LIN {X 0,Y 516.297,Z 411,A -85,B 0,C 180,E1 -4976.05,E2 -4976.05} C_VEL
LIN {X 0,Y 516.258,Z 415.654,A -85,B 0,C 180,E1 -4979.178,E2 -4979.178} C_VEL
LIN {X 0,Y 518.505,Z 428.002,A -85,B 0,C 180,E1 -4979.573,E2 -4979.573} C_VEL
LIN {X 0,Y 518.179,Z 441.043,A -85,B 0,C 180,E1 -4980.07,E2 -4980.07} C_VEL
LIN {X 0,Y 517.831,Z 453.233,A -85,B 0,C 180,E1 -4980.706,E2 -4980.706} C_VEL
LIN {X 0,Y 517.537,Z 464.053,A -85,B 0,C 180,E1 -4981.439,E2 -4981.439} C_VEL
LIN {X 0,Y 517.275,Z 474.235,A -85,B 0,C 180,E1 -4982.296,E2 -4982.296} C_VEL
LIN {X 0,Y 517.004,Z 483.822,A -85,B 0,C 180,E1 -4983.287,E2 -4983.287} C_VEL
LIN {X 0,Y 516.786,Z 492.252,A -85,B 0,C 180,E1 -4984.364,E2 -4984.364} C_VEL
LIN {X 0,Y 516.568,Z 499.577,A -85,B 0,C 180,E1 -4985.517,E2 -4985.517} C_VEL
LIN {X 0,Y 516.456,Z 505.994,A -85,B 0,C 180,E1 -4986.78,E2 -4986.78} C_VEL
LIN {X 0,Y 516.319,Z 511.794,A -85,B 0,C 180,E1 -4988.286,E2 -4988.286} C_VEL
LIN {X 0,Y 516.251,Z 515.814,A -85,B 0,C 180,E1 -4989.779,E2 -4989.779} C_VEL
LIN {X 0,Y 516.155,Z 517.667,A -85,B 0,C 180,E1 -4990.811,E2 -4990.811} C_VEL
LIN {X 0,Y 516.152,Z 518.842,A -85,B 0,C 180,E1 -4991.85,E2 -4991.85} C_VEL
LIN {X 0,Y 516.165,Z 519.286,A -85,B 0,C 180,E1 -4992.905,E2 -4992.905} C_VEL
LIN {X 0,Y 516.188,Z 519.003,A -85,B 0,C 180,E1 -4993.977,E2 -4993.977} C_VEL
LIN {X 0,Y 516.207,Z 517.97,A -85,B 0,C 180,E1 -4995.069,E2 -4995.069} C_VEL
LIN {X 0,Y 516.243,Z 516.116,A -85,B 0,C 180,E1 -4996.18,E2 -4996.18} C_VEL
LIN {X 0,Y 516.328,Z 512.006,A -85,B 0,C 180,E1 -4997.742,E2 -4997.742} C_VEL
LIN {X 0,Y 516.397,Z 508.021,A -85,B 0,C 180,E1 -4998.841,E2 -4998.841} C_VEL
LIN {X 0,Y 516.486,Z 502.965,A -85,B 0,C 180,E1 -4999.95,E2 -4999.95} C_VEL
LIN {X 0,Y 516.683,Z 495.416,A -85,B 0,C 180,E1 -5001.266,E2 -5001.266} C_VEL
LIN {X 0,Y 516.927,Z 487.189,A -85,B 0,C 180,E1 -5002.403,E2 -5002.403} C_VEL
LIN {X 0,Y 517.166,Z 478.617,A -85,B 0,C 180,E1 -5003.37,E2 -5003.37} C_VEL
LIN {X 0,Y 517.497,Z 467.836,A -85,B 0,C 180,E1 -5004.359,E2 -5004.359} C_VEL
LIN {X 0,Y 517.785,Z 457.319,A -85,B 0,C 180,E1 -5005.131,E2 -5005.131} C_VEL
LIN {X 0,Y 518.033,Z 446.537,A -85,B 0,C 180,E1 -5005.759,E2 -5005.759} C_VEL
LIN {X 0,Y 518.35,Z 433.197,A -85,B 0,C 180,E1 -5006.344,E2 -5006.344} C_VEL
LIN {X 0,Y 518.298,Z 426.521,A -85,B 0,C 180,E1 -5006.574,E2 -5006.574} C_VEL
LIN {X 0,Y 516.299,Z 415.747,A -85,B 0,C 180,E1 -5006.923,E2 -5006.923} C_VEL
LIN {X 0,Y 516.306,Z 411.528,A -85,B 0,C 180,E1 -5009.758,E2 -5009.758} C_VEL
LIN {X 0,Y 516.434,Z 407.634,A -85,B 0,C 180,E1 -5012.439,E2 -5012.439} C_VEL
LIN {X 0,Y 516.475,Z 403.919,A -85,B 0,C 180,E1 -5015.049,E2 -5015.049} C_VEL
LIN {X 0,Y 516.543,Z 400.144,A -85,B 0,C 180,E1 -5017.696,E2 -5017.696} C_VEL
LIN {X 0,Y 516.649,Z 396.744,A -85,B 0,C 180,E1 -5020.118,E2 -5020.118} C_VEL
LIN {X 0,Y 516.675,Z 393.324,A -85,B 0,C 180,E1 -5022.587,E2 -5022.587} C_VEL
LIN {X 0,Y 516.733,Z 388.827,A -85,B 0,C 180,E1 -5025.829,E2 -5025.829} C_VEL
LIN {X 0,Y 516.781,Z 386.668,A -85,B 0,C 180,E1 -5027.432,E2 -5027.432} C_VEL
LIN {X 0,Y 516.874,Z 386.105,A -85,B 0,C 180,E1 -5028.232,E2 -5028.232} C_VEL
LIN {X 0,Y 516.968,Z 386.095,A -85,B 0,C 180,E1 -5031.4,E2 -5031.4} C_VEL
LIN {X 0,Y 517.006,Z 386.087,A -85,B 0,C 180,E1 -5033.757,E2 -5033.757} C_VEL
LIN {X 0,Y 517.079,Z 386.08,A -85,B 0,C 180,E1 -5037.663,E2 -5037.663} C_VEL
LIN {X 0,Y 517.092,Z 386.078,A -85,B 0,C 180,E1 -5040.779,E2 -5040.779} C_VEL
LIN {X 0,Y 517.01,Z 386.086,A -85,B 0,C 180,E1 -5043.117,E2 -5043.117} C_VEL
LIN {X 0,Y 517.008,Z 386.087,A -85,B 0,C 180,E1 -5046.243,E2 -5046.243} C_VEL
LIN {X 0,Y 516.951,Z 386.093,A -85,B 0,C 180,E1 -5049.389,E2 -5049.389} C_VEL
LIN {X 0,Y 516.948,Z 386.094,A -85,B 0,C 180,E1 -5051.808,E2 -5051.808} C_VEL
LIN {X 0,Y 516.94,Z 386.096,A -85,B 0,C 180,E1 -5055.147,E2 -5055.147} C_VEL
LIN {X 0,Y 516.922,Z 386.098,A -85,B 0,C 180,E1 -5058.222,E2 -5058.222} C_VEL
LIN {X 0,Y 516.91,Z 386.099,A -85,B 0,C 180,E1 -5060.702,E2 -5060.702} C_VEL
LIN {X 0,Y 516.908,Z 386.097,A -85,B 0,C 180,E1 -5064.072,E2 -5064.072} C_VEL
LIN {X 0,Y 516.926,Z 386.098,A -85,B 0,C 180,E1 -5066.658,E2 -5066.658} C_VEL
LIN {X 0,Y 516.922,Z 386.097,A -85,B 0,C 180,E1 -5069.527,E2 -5069.527} C_VEL
LIN {X 0,Y 516.895,Z 386.1,A -85,B 0,C 180,E1 -5072.544,E2 -5072.544} C_VEL
LIN {X 0,Y 516.878,Z 386.103,A -85,B 0,C 180,E1 -5075.333,E2 -5075.333} C_VEL
LIN {X 0,Y 516.88,Z 386.104,A -85,B 0,C 180,E1 -5077.944,E2 -5077.944} C_VEL
LIN {X 0,Y 516.902,Z 386.1,A -85,B 0,C 180,E1 -5080.74,E2 -5080.74} C_VEL
LIN {X 0,Y 516.881,Z 386.103,A -85,B 0,C 180,E1 -5083.904,E2 -5083.904} C_VEL
LIN {X 0,Y 516.88,Z 386.102,A -85,B 0,C 180,E1 -5086.108,E2 -5086.108} C_VEL
LIN {X 0,Y 516.903,Z 386.1,A -85,B 0,C 180,E1 -5089.261,E2 -5089.261} C_VEL
LIN {X 0,Y 516.918,Z 386.26,A -85,B 0,C 180,E1 -5091.913,E2 -5091.913} C_VEL
LIN {X 0,Y 517.626,Z 390.379,A -85,B 0,C 180,E1 -5093.8,E2 -5093.8} C_VEL
LIN {X 0,Y 517.687,Z 395.366,A -85,B 0,C 180,E1 -5095.907,E2 -5095.907} C_VEL
LIN {X 0,Y 517.366,Z 402.877,A -85,B 0,C 180,E1 -5098.923,E2 -5098.923} C_VEL
LIN {X 0,Y 517.163,Z 409.885,A -85,B 0,C 180,E1 -5101.6,E2 -5101.6} C_VEL
LIN {X 0,Y 516.952,Z 418.116,A -85,B 0,C 180,E1 -5104.644,E2 -5104.644} C_VEL
LIN {X 0,Y 516.833,Z 426.501,A -85,B 0,C 180,E1 -5107.62,E2 -5107.62} C_VEL
LIN {X 0,Y 516.682,Z 434.848,A -85,B 0,C 180,E1 -5110.534,E2 -5110.534} C_VEL
LIN {X 0,Y 516.553,Z 443.402,A -85,B 0,C 180,E1 -5113.399,E2 -5113.399} C_VEL
LIN {X 0,Y 516.494,Z 451.498,A -85,B 0,C 180,E1 -5116.099,E2 -5116.099} C_VEL
LIN {X 0,Y 518.453,Z 465.116,A -85,B 0,C 180,E1 -5116.477,E2 -5116.477} C_VEL
LIN {X 0,Y 518.192,Z 477.346,A -85,B 0,C 180,E1 -5116.92,E2 -5116.92} C_VEL
LIN {X 0,Y 517.871,Z 489.784,A -85,B 0,C 180,E1 -5117.534,E2 -5117.534} C_VEL
LIN {X 0,Y 517.617,Z 500.953,A -85,B 0,C 180,E1 -5118.249,E2 -5118.249} C_VEL
LIN {X 0,Y 517.316,Z 511.907,A -85,B 0,C 180,E1 -5119.135,E2 -5119.135} C_VEL
LIN {X 0,Y 517.003,Z 520.836,A -85,B 0,C 180,E1 -5120.019,E2 -5120.019} C_VEL
LIN {X 0,Y 516.755,Z 530.543,A -85,B 0,C 180,E1 -5121.199,E2 -5121.199} C_VEL
LIN {X 0,Y 516.562,Z 538.27,A -85,B 0,C 180,E1 -5122.377,E2 -5122.377} C_VEL
LIN {X 0,Y 516.427,Z 545.391,A -85,B 0,C 180,E1 -5123.75,E2 -5123.75} C_VEL
LIN {X 0,Y 516.313,Z 550.128,A -85,B 0,C 180,E1 -5124.924,E2 -5124.924} C_VEL
LIN {X 0,Y 516.355,Z 553.751,A -85,B 0,C 180,E1 -5126.098,E2 -5126.098} C_VEL
LIN {X 0,Y 516.282,Z 555.616,A -85,B 0,C 180,E1 -5126.879,E2 -5126.879} C_VEL
LIN {X 0,Y 516.261,Z 557.015,A -85,B 0,C 180,E1 -5127.66,E2 -5127.66} C_VEL
LIN {X 0,Y 516.16,Z 558.621,A -85,B 0,C 180,E1 -5129.22,E2 -5129.22} C_VEL
LIN {X 0,Y 516.154,Z 558.838,A -85,B 0,C 180,E1 -5130,E2 -5130} C_VEL
LIN {X 0,Y 516.192,Z 558.015,A -85,B 0,C 180,E1 -5131.561,E2 -5131.561} C_VEL
LIN {X 0,Y 516.261,Z 557.021,A -85,B 0,C 180,E1 -5132.341,E2 -5132.341} C_VEL
LIN {X 0,Y 516.282,Z 555.624,A -85,B 0,C 180,E1 -5133.122,E2 -5133.122} C_VEL
LIN {X 0,Y 516.326,Z 552.683,A -85,B 0,C 180,E1 -5134.294,E2 -5134.294} C_VEL
LIN {X 0,Y 516.383,Z 548.702,A -85,B 0,C 180,E1 -5135.467,E2 -5135.467} C_VEL
LIN {X 0,Y 516.465,Z 543.401,A -85,B 0,C 180,E1 -5136.679,E2 -5136.679} C_VEL
LIN {X 0,Y 516.598,Z 537.125,A -85,B 0,C 180,E1 -5137.819,E2 -5137.819} C_VEL
LIN {X 0,Y 516.807,Z 529.078,A -85,B 0,C 180,E1 -5138.997,E2 -5138.997} C_VEL
LIN {X 0,Y 516.999,Z 520.876,A -85,B 0,C 180,E1 -5139.981,E2 -5139.981} C_VEL
LIN {X 0,Y 517.318,Z 510.879,A -85,B 0,C 180,E1 -5140.964,E2 -5140.964} C_VEL
LIN {X 0,Y 517.612,Z 501.016,A -85,B 0,C 180,E1 -5141.752,E2 -5141.752} C_VEL
LIN {X 0,Y 517.849,Z 489.862,A -85,B 0,C 180,E1 -5142.467,E2 -5142.467} C_VEL
LIN {X 0,Y 518.17,Z 477.41,A -85,B 0,C 180,E1 -5143.082,E2 -5143.082} C_VEL
LIN {X 0,Y 518.465,Z 464.339,A -85,B 0,C 180,E1 -5143.548,E2 -5143.548} C_VEL
LIN {X 0,Y 516.493,Z 451.65,A -85,B 0,C 180,E1 -5143.902,E2 -5143.902} C_VEL
LIN {X 0,Y 516.597,Z 442.444,A -85,B 0,C 180,E1 -5147.008,E2 -5147.008} C_VEL
LIN {X 0,Y 516.704,Z 433.963,A -85,B 0,C 180,E1 -5149.879,E2 -5149.879} C_VEL
LIN {X 0,Y 516.859,Z 425.579,A -85,B 0,C 180,E1 -5152.801,E2 -5152.801} C_VEL
LIN {X 0,Y 517.023,Z 417.316,A -85,B 0,C 180,E1 -5155.784,E2 -5155.784} C_VEL
LIN {X 0,Y 517.18,Z 410.238,A -85,B 0,C 180,E1 -5158.4,E2 -5158.4} C_VEL
LIN {X 0,Y 517.389,Z 403.001,A -85,B 0,C 180,E1 -5161.155,E2 -5161.155} C_VEL
LIN {X 0,Y 517.701,Z 395.519,A -85,B 0,C 180,E1 -5164.096,E2 -5164.096} C_VEL
LIN {X 0,Y 517.747,Z 391.578,A -85,B 0,C 180,E1 -5165.711,E2 -5165.711} C_VEL
LIN {X 0,Y 516.892,Z 386.102,A -85,B 0,C 180,E1 -5168.088,E2 -5168.088} C_VEL
LIN {X 0,Y 516.886,Z 386.102,A -85,B 0,C 180,E1 -5170.741,E2 -5170.741} C_VEL
LIN {X 0,Y 516.884,Z 386.101,A -85,B 0,C 180,E1 -5172.831,E2 -5172.831} C_VEL
LIN {X 0,Y 516.896,Z 386.101,A -85,B 0,C 180,E1 -5175.007,E2 -5175.007} C_VEL
LIN {X 0,Y 516.914,Z 386.098,A -85,B 0,C 180,E1 -5178.399,E2 -5178.399} C_VEL
LIN {X 0,Y 516.882,Z 386.101,A -85,B 0,C 180,E1 -5181.284,E2 -5181.284} C_VEL
LIN {X 0,Y 516.887,Z 386.101,A -85,B 0,C 180,E1 -5184.221,E2 -5184.221} C_VEL
LIN {X 0,Y 516.895,Z 386.1,A -85,B 0,C 180,E1 -5187.457,E2 -5187.457} C_VEL
LIN {X 0,Y 516.922,Z 386.096,A -85,B 0,C 180,E1 -5190.695,E2 -5190.695} C_VEL
LIN {X 0,Y 516.943,Z 386.095,A -85,B 0,C 180,E1 -5193.804,E2 -5193.804} C_VEL
LIN {X 0,Y 516.866,Z 386.103,A -85,B 0,C 180,E1 -5196.776,E2 -5196.776} C_VEL
LIN {X 0,Y 516.94,Z 386.095,A -85,B 0,C 180,E1 -5199.732,E2 -5199.732} C_VEL
LIN {X 0,Y 516.922,Z 386.096,A -85,B 0,C 180,E1 -5202.596,E2 -5202.596} C_VEL
LIN {X 0,Y 516.943,Z 386.094,A -85,B 0,C 180,E1 -5205.03,E2 -5205.03} C_VEL
LIN {X 0,Y 516.966,Z 386.092,A -85,B 0,C 180,E1 -5208.234,E2 -5208.234} C_VEL
LIN {X 0,Y 516.97,Z 386.091,A -85,B 0,C 180,E1 -5211.4,E2 -5211.4} C_VEL
LIN {X 0,Y 517.011,Z 386.086,A -85,B 0,C 180,E1 -5213.757,E2 -5213.757} C_VEL
LIN {X 0,Y 517.082,Z 386.077,A -85,B 0,C 180,E1 -5217.663,E2 -5217.663} C_VEL
LIN {X 0,Y 517.093,Z 386.075,A -85,B 0,C 180,E1 -5220.779,E2 -5220.779} C_VEL
LIN {X 0,Y 517.014,Z 386.085,A -85,B 0,C 180,E1 -5223.117,E2 -5223.117} C_VEL
LIN {X 0,Y 517.011,Z 386.087,A -85,B 0,C 180,E1 -5226.243,E2 -5226.243} C_VEL
LIN {X 0,Y 516.953,Z 386.094,A -85,B 0,C 180,E1 -5229.389,E2 -5229.389} C_VEL
LIN {X 0,Y 516.952,Z 386.093,A -85,B 0,C 180,E1 -5231.807,E2 -5231.807} C_VEL
LIN {X 0,Y 516.945,Z 386.094,A -85,B 0,C 180,E1 -5235.146,E2 -5235.146} C_VEL
LIN {X 0,Y 516.926,Z 386.097,A -85,B 0,C 180,E1 -5238.222,E2 -5238.222} C_VEL
LIN {X 0,Y 516.912,Z 386.098,A -85,B 0,C 180,E1 -5240.701,E2 -5240.701} C_VEL
LIN {X 0,Y 516.904,Z 386.1,A -85,B 0,C 180,E1 -5244.072,E2 -5244.072} C_VEL
LIN {X 0,Y 516.926,Z 386.096,A -85,B 0,C 180,E1 -5246.658,E2 -5246.658} C_VEL
LIN {X 0,Y 516.911,Z 386.098,A -85,B 0,C 180,E1 -5249.524,E2 -5249.524} C_VEL
LIN {X 0,Y 516.898,Z 386.1,A -85,B 0,C 180,E1 -5252.544,E2 -5252.544} C_VEL
LIN {X 0,Y 516.881,Z 386.101,A -85,B 0,C 180,E1 -5255.332,E2 -5255.332} C_VEL
LIN {X 0,Y 516.882,Z 386.101,A -85,B 0,C 180,E1 -5257.943,E2 -5257.943} C_VEL
LIN {X 0,Y 516.883,Z 386.103,A -85,B 0,C 180,E1 -5260.742,E2 -5260.742} C_VEL
LIN {X 0,Y 516.885,Z 386.103,A -85,B 0,C 180,E1 -5262.831,E2 -5262.831} C_VEL
LIN {X 0,Y 516.896,Z 386.1,A -85,B 0,C 180,E1 -5265.007,E2 -5265.007} C_VEL
LIN {X 0,Y 516.918,Z 386.097,A -85,B 0,C 180,E1 -5268.398,E2 -5268.398} C_VEL
LIN {X 0,Y 516.882,Z 386.103,A -85,B 0,C 180,E1 -5270.296,E2 -5270.296} C_VEL
LIN {X 0,Y 516.211,Z 386.186,A -85,B 0,C 180,E1 -5270.946,E2 -5270.946} C_VEL
LIN {X 0,Y 513.366,Z 386.54,A -85,B 0,C 180,E1 -5272.002,E2 -5272.002} C_VEL
LIN {X 0,Y 510.96,Z 386.841,A -85,B 0,C 180,E1 -5272.852,E2 -5272.852} C_VEL
LIN {X 0,Y 509.92,Z 386.97,A -85,B 0,C 180,E1 -5273.509,E2 -5273.509} C_VEL
LIN {X 0,Y 509.832,Z 386.979,A -85,B 0,C 180,E1 -5273.731,E2 -5273.731} C_VEL
LIN {X 0,Y 509.862,Z 386.976,A -85,B 0,C 180,E1 -5276.539,E2 -5276.539} C_VEL
LIN {X 0,Y 509.847,Z 386.978,A -85,B 0,C 180,E1 -5279.334,E2 -5279.334} C_VEL
LIN {X 0,Y 509.894,Z 386.973,A -85,B 0,C 180,E1 -5282.054,E2 -5282.054} C_VEL
LIN {X 0,Y 509.879,Z 386.974,A -85,B 0,C 180,E1 -5284.704,E2 -5284.704} C_VEL
LIN {X 0,Y 509.829,Z 386.978,A -85,B 0,C 180,E1 -5287.458,E2 -5287.458} C_VEL
LIN {X 0,Y 509.919,Z 386.968,A -85,B 0,C 180,E1 -5289.845,E2 -5289.845} C_VEL
LIN {X 0,Y 509.881,Z 386.972,A -85,B 0,C 180,E1 -5293.174,E2 -5293.174} C_VEL
LIN {X 0,Y 509.866,Z 386.975,A -85,B 0,C 180,E1 -5295.634,E2 -5295.634} C_VEL
LIN {X 0,Y 509.915,Z 386.969,A -85,B 0,C 180,E1 -5298.874,E2 -5298.874} C_VEL
LIN {X 0,Y 509.953,Z 386.965,A -85,B 0,C 180,E1 -5302.078,E2 -5302.078} C_VEL
LIN {X 0,Y 509.984,Z 386.962,A -85,B 0,C 180,E1 -5304.464,E2 -5304.464} C_VEL
LIN {X 0,Y 510.058,Z 386.951,A -85,B 0,C 180,E1 -5307.631,E2 -5307.631} C_VEL
LIN {X 0,Y 510.066,Z 386.951,A -85,B 0,C 180,E1 -5310.789,E2 -5310.789} C_VEL
LIN {X 0,Y 509.956,Z 386.964,A -85,B 0,C 180,E1 -5313.16,E2 -5313.16} C_VEL
LIN {X 0,Y 509.938,Z 386.967,A -85,B 0,C 180,E1 -5316.33,E2 -5316.33} C_VEL
LIN {X 0,Y 509.706,Z 386.998,A -85,B 0,C 180,E1 -5318.723,E2 -5318.723} C_VEL
LIN {X 0,Y 509.616,Z 391.348,A -85,B 0,C 180,E1 -5321.938,E2 -5321.938} C_VEL
LIN {X 0,Y 509.499,Z 395.893,A -85,B 0,C 180,E1 -5325.193,E2 -5325.193} C_VEL
LIN {X 0,Y 509.404,Z 400.582,A -85,B 0,C 180,E1 -5328.5,E2 -5328.5} C_VEL
LIN {X 0,Y 509.281,Z 404.229,A -85,B 0,C 180,E1 -5331.026,E2 -5331.026} C_VEL
LIN {X 0,Y 509.258,Z 407.951,A -85,B 0,C 180,E1 -5333.591,E2 -5333.591} C_VEL
LIN {X 0,Y 509.213,Z 411.861,A -85,B 0,C 180,E1 -5336.219,E2 -5336.219} C_VEL
LIN {X 0,Y 509.193,Z 416.037,A -85,B 0,C 180,E1 -5338.997,E2 -5338.997} C_VEL
LIN {X 0,Y 511.576,Z 428.689,A -85,B 0,C 180,E1 -5339.404,E2 -5339.404} C_VEL
LIN {X 0,Y 511.235,Z 441.825,A -85,B 0,C 180,E1 -5339.916,E2 -5339.916} C_VEL
LIN {X 0,Y 510.919,Z 453.048,A -85,B 0,C 180,E1 -5340.511,E2 -5340.511} C_VEL
LIN {X 0,Y 510.566,Z 464.641,A -85,B 0,C 180,E1 -5341.307,E2 -5341.307} C_VEL
LIN {X 0,Y 510.273,Z 475.615,A -85,B 0,C 180,E1 -5342.255,E2 -5342.255} C_VEL
LIN {X 0,Y 509.992,Z 485.086,A -85,B 0,C 180,E1 -5343.275,E2 -5343.275} C_VEL
LIN {X 0,Y 509.718,Z 493.709,A -85,B 0,C 180,E1 -5344.423,E2 -5344.423} C_VEL
LIN {X 0,Y 509.497,Z 501.397,A -85,B 0,C 180,E1 -5345.694,E2 -5345.694} C_VEL
LIN {X 0,Y 509.314,Z 507.926,A -85,B 0,C 180,E1 -5347.087,E2 -5347.087} C_VEL
LIN {X 0,Y 509.235,Z 512.588,A -85,B 0,C 180,E1 -5348.392,E2 -5348.392} C_VEL
LIN {X 0,Y 509.14,Z 516.501,A -85,B 0,C 180,E1 -5349.931,E2 -5349.931} C_VEL
LIN {X 0,Y 509.058,Z 518.806,A -85,B 0,C 180,E1 -5351.504,E2 -5351.504} C_VEL
LIN {X 0,Y 509.079,Z 519.572,A -85,B 0,C 180,E1 -5352.972,E2 -5352.972} C_VEL
LIN {X 0,Y 509.105,Z 519.195,A -85,B 0,C 180,E1 -5354.123,E2 -5354.123} C_VEL
LIN {X 0,Y 509.121,Z 518.028,A -85,B 0,C 180,E1 -5355.25,E2 -5355.25} C_VEL
LIN {X 0,Y 509.173,Z 516.09,A -85,B 0,C 180,E1 -5356.359,E2 -5356.359} C_VEL
LIN {X 0,Y 509.271,Z 512.167,A -85,B 0,C 180,E1 -5357.843,E2 -5357.843} C_VEL
LIN {X 0,Y 509.324,Z 508.083,A -85,B 0,C 180,E1 -5358.974,E2 -5358.974} C_VEL
LIN {X 0,Y 509.487,Z 501.648,A -85,B 0,C 180,E1 -5360.359,E2 -5360.359} C_VEL
LIN {X 0,Y 509.705,Z 493.893,A -85,B 0,C 180,E1 -5361.649,E2 -5361.649} C_VEL
LIN {X 0,Y 509.967,Z 486.313,A -85,B 0,C 180,E1 -5362.672,E2 -5362.672} C_VEL
LIN {X 0,Y 510.244,Z 477.233,A -85,B 0,C 180,E1 -5363.681,E2 -5363.681} C_VEL
LIN {X 0,Y 510.569,Z 467.144,A -85,B 0,C 180,E1 -5364.594,E2 -5364.594} C_VEL
LIN {X 0,Y 510.863,Z 456.701,A -85,B 0,C 180,E1 -5365.352,E2 -5365.352} C_VEL
LIN {X 0,Y 511.157,Z 444.61,A -85,B 0,C 180,E1 -5366.044,E2 -5366.044} C_VEL
LIN {X 0,Y 511.464,Z 433.096,A -85,B 0,C 180,E1 -5366.54,E2 -5366.54} C_VEL
LIN {X 0,Y 511.261,Z 426.599,A -85,B 0,C 180,E1 -5366.768,E2 -5366.768} C_VEL
LIN {X 0,Y 509.233,Z 416.078,A -85,B 0,C 180,E1 -5367.1,E2 -5367.1} C_VEL
LIN {X 0,Y 509.269,Z 411.267,A -85,B 0,C 180,E1 -5370.389,E2 -5370.389} C_VEL
LIN {X 0,Y 509.34,Z 407.659,A -85,B 0,C 180,E1 -5372.913,E2 -5372.913} C_VEL
LIN {X 0,Y 509.413,Z 403.837,A -85,B 0,C 180,E1 -5375.58,E2 -5375.58} C_VEL
LIN {X 0,Y 509.486,Z 400.261,A -85,B 0,C 180,E1 -5378.133,E2 -5378.133} C_VEL
LIN {X 0,Y 509.561,Z 396.743,A -85,B 0,C 180,E1 -5380.67,E2 -5380.67} C_VEL
LIN {X 0,Y 509.604,Z 393.284,A -85,B 0,C 180,E1 -5383.165,E2 -5383.165} C_VEL
LIN {X 0,Y 509.698,Z 389.968,A -85,B 0,C 180,E1 -5385.629,E2 -5385.629} C_VEL
LIN {X 0,Y 509.722,Z 387.777,A -85,B 0,C 180,E1 -5387.255,E2 -5387.255} C_VEL
LIN {X 0,Y 509.822,Z 386.984,A -85,B 0,C 180,E1 -5388.164,E2 -5388.164} C_VEL
LIN {X 0,Y 509.914,Z 386.974,A -85,B 0,C 180,E1 -5391.28,E2 -5391.28} C_VEL
LIN {X 0,Y 509.974,Z 386.963,A -85,B 0,C 180,E1 -5393.67,E2 -5393.67} C_VEL
LIN {X 0,Y 510.051,Z 386.955,A -85,B 0,C 180,E1 -5397.631,E2 -5397.631} C_VEL
LIN {X 0,Y 510.062,Z 386.953,A -85,B 0,C 180,E1 -5400.79,E2 -5400.79} C_VEL
LIN {X 0,Y 509.952,Z 386.965,A -85,B 0,C 180,E1 -5403.16,E2 -5403.16} C_VEL
LIN {X 0,Y 509.976,Z 386.962,A -85,B 0,C 180,E1 -5406.33,E2 -5406.33} C_VEL
LIN {X 0,Y 509.912,Z 386.97,A -85,B 0,C 180,E1 -5408.72,E2 -5408.72} C_VEL
LIN {X 0,Y 509.9,Z 386.972,A -85,B 0,C 180,E1 -5411.932,E2 -5411.932} C_VEL
LIN {X 0,Y 509.889,Z 386.975,A -85,B 0,C 180,E1 -5415.242,E2 -5415.242} C_VEL
LIN {X 0,Y 509.885,Z 386.973,A -85,B 0,C 180,E1 -5418.001,E2 -5418.001} C_VEL
LIN {X 0,Y 509.848,Z 386.978,A -85,B 0,C 180,E1 -5421.002,E2 -5421.002} C_VEL
LIN {X 0,Y 509.833,Z 386.981,A -85,B 0,C 180,E1 -5423.563,E2 -5423.563} C_VEL
LIN {X 0,Y 509.91,Z 386.97,A -85,B 0,C 180,E1 -5426.38,E2 -5426.38} C_VEL
LIN {X 0,Y 509.883,Z 386.976,A -85,B 0,C 180,E1 -5428.844,E2 -5428.844} C_VEL
LIN {X 0,Y 509.819,Z 386.982,A -85,B 0,C 180,E1 -5431.59,E2 -5431.59} C_VEL
LIN {X 0,Y 509.85,Z 386.978,A -85,B 0,C 180,E1 -5434.414,E2 -5434.414} C_VEL
LIN {X 0,Y 509.817,Z 386.984,A -85,B 0,C 180,E1 -5437.341,E2 -5437.341} C_VEL
LIN {X 0,Y 509.86,Z 386.979,A -85,B 0,C 180,E1 -5440.38,E2 -5440.38} C_VEL
LIN {X 0,Y 509.822,Z 386.982,A -85,B 0,C 180,E1 -5443.063,E2 -5443.063} C_VEL
LIN {X 0,Y 509.828,Z 386.981,A -85,B 0,C 180,E1 -5445.793,E2 -5445.793} C_VEL
LIN {X 0,Y 509.865,Z 386.975,A -85,B 0,C 180,E1 -5448.576,E2 -5448.576} C_VEL
LIN {X 0,Y 509.854,Z 387.091,A -85,B 0,C 180,E1 -5451.663,E2 -5451.663} C_VEL
LIN {X 0,Y 510.636,Z 391.477,A -85,B 0,C 180,E1 -5453.715,E2 -5453.715} C_VEL
LIN {X 0,Y 510.706,Z 395.971,A -85,B 0,C 180,E1 -5455.658,E2 -5455.658} C_VEL
LIN {X 0,Y 510.391,Z 403.245,A -85,B 0,C 180,E1 -5458.62,E2 -5458.62} C_VEL
LIN {X 0,Y 510.167,Z 409.74,A -85,B 0,C 180,E1 -5461.174,E2 -5461.174} C_VEL
LIN {X 0,Y 509.949,Z 417.958,A -85,B 0,C 180,E1 -5464.271,E2 -5464.271} C_VEL
LIN {X 0,Y 509.778,Z 426.769,A -85,B 0,C 180,E1 -5467.472,E2 -5467.472} C_VEL
LIN {X 0,Y 509.609,Z 434.653,A -85,B 0,C 180,E1 -5470.253,E2 -5470.253} C_VEL
LIN {X 0,Y 509.485,Z 443.148,A -85,B 0,C 180,E1 -5473.162,E2 -5473.162} C_VEL
LIN {X 0,Y 509.395,Z 451.195,A -85,B 0,C 180,E1 -5475.901,E2 -5475.901} C_VEL
LIN {X 0,Y 511.524,Z 465.534,A -85,B 0,C 180,E1 -5476.316,E2 -5476.316} C_VEL
LIN {X 0,Y 511.24,Z 478.133,A -85,B 0,C 180,E1 -5476.789,E2 -5476.789} C_VEL
LIN {X 0,Y 510.887,Z 490.799,A -85,B 0,C 180,E1 -5477.438,E2 -5477.438} C_VEL
LIN {X 0,Y 510.605,Z 501.947,A -85,B 0,C 180,E1 -5478.186,E2 -5478.186} C_VEL
LIN {X 0,Y 510.285,Z 512.66,A -85,B 0,C 180,E1 -5479.084,E2 -5479.084} C_VEL
LIN {X 0,Y 509.937,Z 522.316,A -85,B 0,C 180,E1 -5480.08,E2 -5480.08} C_VEL
LIN {X 0,Y 509.703,Z 530.235,A -85,B 0,C 180,E1 -5481.077,E2 -5481.077} C_VEL
LIN {X 0,Y 509.494,Z 537.971,A -85,B 0,C 180,E1 -5482.271,E2 -5482.271} C_VEL
LIN {X 0,Y 509.326,Z 545.098,A -85,B 0,C 180,E1 -5483.663,E2 -5483.663} C_VEL
LIN {X 0,Y 509.245,Z 549.842,A -85,B 0,C 180,E1 -5484.854,E2 -5484.854} C_VEL
LIN {X 0,Y 509.25,Z 553.468,A -85,B 0,C 180,E1 -5486.044,E2 -5486.044} C_VEL
LIN {X 0,Y 509.2,Z 555.338,A -85,B 0,C 180,E1 -5486.836,E2 -5486.836} C_VEL
LIN {X 0,Y 509.19,Z 556.74,A -85,B 0,C 180,E1 -5487.627,E2 -5487.627} C_VEL
LIN {X 0,Y 509.073,Z 558.348,A -85,B 0,C 180,E1 -5489.209,E2 -5489.209} C_VEL
LIN {X 0,Y 509.065,Z 558.567,A -85,B 0,C 180,E1 -5490,E2 -5490} C_VEL
LIN {X 0,Y 509.112,Z 557.745,A -85,B 0,C 180,E1 -5491.582,E2 -5491.582} C_VEL
LIN {X 0,Y 509.19,Z 556.752,A -85,B 0,C 180,E1 -5492.373,E2 -5492.373} C_VEL
LIN {X 0,Y 509.201,Z 555.353,A -85,B 0,C 180,E1 -5493.165,E2 -5493.165} C_VEL
LIN {X 0,Y 509.216,Z 552.411,A -85,B 0,C 180,E1 -5494.354,E2 -5494.354} C_VEL
LIN {X 0,Y 509.305,Z 548.43,A -85,B 0,C 180,E1 -5495.543,E2 -5495.543} C_VEL
LIN {X 0,Y 509.402,Z 542.757,A -85,B 0,C 180,E1 -5496.845,E2 -5496.845} C_VEL
LIN {X 0,Y 509.563,Z 535.606,A -85,B 0,C 180,E1 -5498.127,E2 -5498.127} C_VEL
LIN {X 0,Y 509.793,Z 527.301,A -85,B 0,C 180,E1 -5499.322,E2 -5499.322} C_VEL
LIN {X 0,Y 510.013,Z 518.782,A -85,B 0,C 180,E1 -5500.32,E2 -5500.32} C_VEL
LIN {X 0,Y 510.406,Z 508.264,A -85,B 0,C 180,E1 -5501.316,E2 -5501.316} C_VEL
LIN {X 0,Y 510.66,Z 497.108,A -85,B 0,C 180,E1 -5502.168,E2 -5502.168} C_VEL
LIN {X 0,Y 511.004,Z 486.461,A -85,B 0,C 180,E1 -5502.813,E2 -5502.813} C_VEL
LIN {X 0,Y 511.327,Z 474.749,A -85,B 0,C 180,E1 -5503.361,E2 -5503.361} C_VEL
LIN {X 0,Y 511.34,Z 463.555,A -85,B 0,C 180,E1 -5503.753,E2 -5503.753} C_VEL
LIN {X 0,Y 509.404,Z 451.39,A -85,B 0,C 180,E1 -5504.099,E2 -5504.099} C_VEL
LIN {X 0,Y 509.499,Z 443.469,A -85,B 0,C 180,E1 -5506.839,E2 -5506.839} C_VEL
LIN {X 0,Y 509.647,Z 434.994,A -85,B 0,C 180,E1 -5509.746,E2 -5509.746} C_VEL
LIN {X 0,Y 509.81,Z 426.62,A -85,B 0,C 180,E1 -5512.706,E2 -5512.706} C_VEL
LIN {X 0,Y 509.985,Z 418.367,A -85,B 0,C 180,E1 -5515.728,E2 -5515.728} C_VEL
LIN {X 0,Y 510.185,Z 410.121,A -85,B 0,C 180,E1 -5518.825,E2 -5518.825} C_VEL
LIN {X 0,Y 510.419,Z 403.092,A -85,B 0,C 180,E1 -5521.549,E2 -5521.549} C_VEL
LIN {X 0,Y 510.73,Z 396.125,A -85,B 0,C 180,E1 -5524.346,E2 -5524.346} C_VEL
LIN {X 0,Y 510.595,Z 391.497,A -85,B 0,C 180,E1 -5526.29,E2 -5526.29} C_VEL
LIN {X 0,Y 509.855,Z 386.978,A -85,B 0,C 180,E1 -5528.338,E2 -5528.338} C_VEL
LIN {X 0,Y 509.859,Z 386.977,A -85,B 0,C 180,E1 -5531.425,E2 -5531.425} C_VEL
LIN {X 0,Y 509.84,Z 386.98,A -85,B 0,C 180,E1 -5534.67,E2 -5534.67} C_VEL
LIN {X 0,Y 509.857,Z 386.977,A -85,B 0,C 180,E1 -5538.103,E2 -5538.103} C_VEL
LIN {X 0,Y 509.847,Z 386.978,A -85,B 0,C 180,E1 -5540.647,E2 -5540.647} C_VEL
LIN {X 0,Y 509.835,Z 386.979,A -85,B 0,C 180,E1 -5543.647,E2 -5543.647} C_VEL
LIN {X 0,Y 509.843,Z 386.978,A -85,B 0,C 180,E1 -5546.538,E2 -5546.538} C_VEL
LIN {X 0,Y 509.846,Z 386.978,A -85,B 0,C 180,E1 -5549.334,E2 -5549.334} C_VEL
LIN {X 0,Y 509.893,Z 386.97,A -85,B 0,C 180,E1 -5552.054,E2 -5552.054} C_VEL
LIN {X 0,Y 509.877,Z 386.974,A -85,B 0,C 180,E1 -5554.704,E2 -5554.704} C_VEL
LIN {X 0,Y 509.827,Z 386.981,A -85,B 0,C 180,E1 -5557.458,E2 -5557.458} C_VEL
LIN {X 0,Y 509.917,Z 386.969,A -85,B 0,C 180,E1 -5559.845,E2 -5559.845} C_VEL
LIN {X 0,Y 509.882,Z 386.975,A -85,B 0,C 180,E1 -5563.175,E2 -5563.175} C_VEL
LIN {X 0,Y 509.864,Z 386.977,A -85,B 0,C 180,E1 -5565.634,E2 -5565.634} C_VEL
LIN {X 0,Y 509.913,Z 386.97,A -85,B 0,C 180,E1 -5568.874,E2 -5568.874} C_VEL
LIN {X 0,Y 509.952,Z 386.964,A -85,B 0,C 180,E1 -5572.078,E2 -5572.078} C_VEL
LIN {X 0,Y 509.982,Z 386.961,A -85,B 0,C 180,E1 -5574.464,E2 -5574.464} C_VEL
LIN {X 0,Y 510.053,Z 386.953,A -85,B 0,C 180,E1 -5577.631,E2 -5577.631} C_VEL
LIN {X 0,Y 510.064,Z 386.951,A -85,B 0,C 180,E1 -5580.789,E2 -5580.789} C_VEL
LIN {X 0,Y 509.956,Z 386.964,A -85,B 0,C 180,E1 -5583.16,E2 -5583.16} C_VEL
LIN {X 0,Y 509.979,Z 386.962,A -85,B 0,C 180,E1 -5586.33,E2 -5586.33} C_VEL
LIN {X 0,Y 509.916,Z 386.97,A -85,B 0,C 180,E1 -5588.72,E2 -5588.72} C_VEL
LIN {X 0,Y 509.905,Z 386.971,A -85,B 0,C 180,E1 -5591.932,E2 -5591.932} C_VEL
LIN {X 0,Y 509.894,Z 386.973,A -85,B 0,C 180,E1 -5595.242,E2 -5595.242} C_VEL
LIN {X 0,Y 509.889,Z 386.973,A -85,B 0,C 180,E1 -5598.001,E2 -5598.001} C_VEL
LIN {X 0,Y 509.85,Z 386.977,A -85,B 0,C 180,E1 -5601.002,E2 -5601.002} C_VEL
LIN {X 0,Y 509.865,Z 386.975,A -85,B 0,C 180,E1 -5604.426,E2 -5604.426} C_VEL
LIN {X 0,Y 509.885,Z 386.973,A -85,B 0,C 180,E1 -5607.056,E2 -5607.056} C_VEL
LIN {X 0,Y 509.858,Z 386.977,A -85,B 0,C 180,E1 -5609.751,E2 -5609.751} C_VEL
LIN {X 0,Y 509.875,Z 386.974,A -85,B 0,C 180,E1 -5612.774,E2 -5612.774} C_VEL
LIN {X 0,Y 509.841,Z 386.979,A -85,B 0,C 180,E1 -5615.581,E2 -5615.581} C_VEL
LIN {X 0,Y 509.851,Z 386.979,A -85,B 0,C 180,E1 -5618.338,E2 -5618.338} C_VEL
LIN {X 0,Y 509.856,Z 386.976,A -85,B 0,C 180,E1 -5621.426,E2 -5621.426} C_VEL
LIN {X 0,Y 509.84,Z 386.979,A -85,B 0,C 180,E1 -5624.67,E2 -5624.67} C_VEL
LIN {X 0,Y 509.86,Z 386.977,A -85,B 0,C 180,E1 -5628.103,E2 -5628.103} C_VEL
LIN {X 0,Y 509.847,Z 386.978,A -85,B 0,C 180,E1 -5630.648,E2 -5630.648} C_VEL
LIN {X 0,Y 509.832,Z 386.979,A -85,B 0,C 180,E1 -5633.731,E2 -5633.731} C_VEL
LIN {X 0,Y 509.165,Z 387.063,A -85,B 0,C 180,E1 -5634.391,E2 -5634.391} C_VEL
LIN {X 0,Y 506.35,Z 387.413,A -85,B 0,C 180,E1 -5635.463,E2 -5635.463} C_VEL
LIN {X 0,Y 503.958,Z 387.713,A -85,B 0,C 180,E1 -5636.326,E2 -5636.326} C_VEL
LIN {X 0,Y 502.908,Z 387.843,A -85,B 0,C 180,E1 -5636.992,E2 -5636.992} C_VEL
LIN {X 0,Y 502.81,Z 387.853,A -85,B 0,C 180,E1 -5637.218,E2 -5637.218} C_VEL
LIN {X 0,Y 502.817,Z 387.854,A -85,B 0,C 180,E1 -5640.065,E2 -5640.065} C_VEL
LIN {X 0,Y 502.834,Z 387.852,A -85,B 0,C 180,E1 -5642.533,E2 -5642.533} C_VEL
LIN {X 0,Y 502.829,Z 387.852,A -85,B 0,C 180,E1 -5645.299,E2 -5645.299} C_VEL
LIN {X 0,Y 502.783,Z 387.857,A -85,B 0,C 180,E1 -5647.826,E2 -5647.826} C_VEL
LIN {X 0,Y 502.827,Z 387.854,A -85,B 0,C 180,E1 -5650.4,E2 -5650.4} C_VEL
LIN {X 0,Y 502.83,Z 387.852,A -85,B 0,C 180,E1 -5652.931,E2 -5652.931} C_VEL
LIN {X 0,Y 502.847,Z 387.85,A -85,B 0,C 180,E1 -5655.429,E2 -5655.429} C_VEL
LIN {X 0,Y 502.879,Z 387.848,A -85,B 0,C 180,E1 -5658.717,E2 -5658.717} C_VEL
LIN {X 0,Y 502.903,Z 387.842,A -85,B 0,C 180,E1 -5661.966,E2 -5661.966} C_VEL
LIN {X 0,Y 502.94,Z 387.839,A -85,B 0,C 180,E1 -5664.386,E2 -5664.386} C_VEL
LIN {X 0,Y 503.027,Z 387.827,A -85,B 0,C 180,E1 -5667.598,E2 -5667.598} C_VEL
LIN {X 0,Y 503.031,Z 387.827,A -85,B 0,C 180,E1 -5670,E2 -5670} C_VEL
LIN {X 0,Y 503.027,Z 387.827,A -85,B 0,C 180,E1 -5672.402,E2 -5672.402} C_VEL
LIN {X 0,Y 502.93,Z 387.841,A -85,B 0,C 180,E1 -5675.613,E2 -5675.613} C_VEL
LIN {X 0,Y 502.774,Z 387.861,A -85,B 0,C 180,E1 -5678.035,E2 -5678.035} C_VEL
LIN {X 0,Y 502.648,Z 387.914,A -85,B 0,C 180,E1 -5678.847,E2 -5678.847} C_VEL
LIN {X 0,Y 502.533,Z 392.335,A -85,B 0,C 180,E1 -5682.109,E2 -5682.109} C_VEL
LIN {X 0,Y 502.409,Z 396.905,A -85,B 0,C 180,E1 -5685.413,E2 -5685.413} C_VEL
LIN {X 0,Y 502.377,Z 400.487,A -85,B 0,C 180,E1 -5687.957,E2 -5687.957} C_VEL
LIN {X 0,Y 502.258,Z 404.074,A -85,B 0,C 180,E1 -5690.476,E2 -5690.476} C_VEL
LIN {X 0,Y 502.192,Z 407.794,A -85,B 0,C 180,E1 -5693.069,E2 -5693.069} C_VEL
LIN {X 0,Y 502.133,Z 411.675,A -85,B 0,C 180,E1 -5695.714,E2 -5695.714} C_VEL
LIN {X 0,Y 502.091,Z 416.19,A -85,B 0,C 180,E1 -5698.789,E2 -5698.789} C_VEL
LIN {X 0,Y 504.551,Z 428.772,A -85,B 0,C 180,E1 -5699.206,E2 -5699.206} C_VEL
LIN {X 0,Y 504.391,Z 441.327,A -85,B 0,C 180,E1 -5699.703,E2 -5699.703} C_VEL
LIN {X 0,Y 503.993,Z 452.989,A -85,B 0,C 180,E1 -5700.32,E2 -5700.32} C_VEL
LIN {X 0,Y 503.665,Z 464.095,A -85,B 0,C 180,E1 -5701.083,E2 -5701.083} C_VEL
LIN {X 0,Y 503.298,Z 475.248,A -85,B 0,C 180,E1 -5702.047,E2 -5702.047} C_VEL
LIN {X 0,Y 503.026,Z 484.521,A -85,B 0,C 180,E1 -5703.04,E2 -5703.04} C_VEL
LIN {X 0,Y 502.709,Z 493.333,A -85,B 0,C 180,E1 -5704.209,E2 -5704.209} C_VEL
LIN {X 0,Y 502.473,Z 500.482,A -85,B 0,C 180,E1 -5705.379,E2 -5705.379} C_VEL
LIN {X 0,Y 502.329,Z 507.085,A -85,B 0,C 180,E1 -5706.734,E2 -5706.734} C_VEL
LIN {X 0,Y 502.187,Z 511.869,A -85,B 0,C 180,E1 -5708.007,E2 -5708.007} C_VEL
LIN {X 0,Y 502.114,Z 514.841,A -85,B 0,C 180,E1 -5709.039,E2 -5709.039} C_VEL
LIN {X 0,Y 502.057,Z 517.12,A -85,B 0,C 180,E1 -5710.084,E2 -5710.084} C_VEL
LIN {X 0,Y 501.96,Z 518.747,A -85,B 0,C 180,E1 -5711.151,E2 -5711.151} C_VEL
LIN {X 0,Y 501.975,Z 519.624,A -85,B 0,C 180,E1 -5712.223,E2 -5712.223} C_VEL
LIN {X 0,Y 501.99,Z 519.805,A -85,B 0,C 180,E1 -5713.315,E2 -5713.315} C_VEL
LIN {X 0,Y 502.035,Z 519.247,A -85,B 0,C 180,E1 -5714.443,E2 -5714.443} C_VEL
LIN {X 0,Y 502.037,Z 517.891,A -85,B 0,C 180,E1 -5715.577,E2 -5715.577} C_VEL
LIN {X 0,Y 502.103,Z 515.703,A -85,B 0,C 180,E1 -5716.706,E2 -5716.706} C_VEL
LIN {X 0,Y 502.208,Z 512.547,A -85,B 0,C 180,E1 -5717.875,E2 -5717.875} C_VEL
LIN {X 0,Y 502.25,Z 508.268,A -85,B 0,C 180,E1 -5719.079,E2 -5719.079} C_VEL
LIN {X 0,Y 502.418,Z 502.751,A -85,B 0,C 180,E1 -5720.295,E2 -5720.295} C_VEL
LIN {X 0,Y 502.646,Z 495.717,A -85,B 0,C 180,E1 -5721.534,E2 -5721.534} C_VEL
LIN {X 0,Y 502.92,Z 487.735,A -85,B 0,C 180,E1 -5722.662,E2 -5722.662} C_VEL
LIN {X 0,Y 503.202,Z 478.62,A -85,B 0,C 180,E1 -5723.713,E2 -5723.713} C_VEL
LIN {X 0,Y 503.568,Z 469.136,A -85,B 0,C 180,E1 -5724.606,E2 -5724.606} C_VEL
LIN {X 0,Y 503.921,Z 457.986,A -85,B 0,C 180,E1 -5725.456,E2 -5725.456} C_VEL
LIN {X 0,Y 504.223,Z 445.821,A -85,B 0,C 180,E1 -5726.175,E2 -5726.175} C_VEL
LIN {X 0,Y 504.58,Z 433.298,A -85,B 0,C 180,E1 -5726.729,E2 -5726.729} C_VEL
LIN {X 0,Y 504.334,Z 427.285,A -85,B 0,C 180,E1 -5726.946,E2 -5726.946} C_VEL
LIN {X 0,Y 502.177,Z 416.372,A -85,B 0,C 180,E1 -5727.307,E2 -5727.307} C_VEL
LIN {X 0,Y 502.183,Z 412.215,A -85,B 0,C 180,E1 -5730.189,E2 -5730.189} C_VEL
LIN {X 0,Y 502.277,Z 407.631,A -85,B 0,C 180,E1 -5733.4,E2 -5733.4} C_VEL
LIN {X 0,Y 502.339,Z 403.877,A -85,B 0,C 180,E1 -5736.063,E2 -5736.063} C_VEL
LIN {X 0,Y 502.441,Z 400.266,A -85,B 0,C 180,E1 -5738.674,E2 -5738.674} C_VEL
LIN {X 0,Y 502.512,Z 396.739,A -85,B 0,C 180,E1 -5741.236,E2 -5741.236} C_VEL
LIN {X 0,Y 502.572,Z 393.32,A -85,B 0,C 180,E1 -5743.759,E2 -5743.759} C_VEL
LIN {X 0,Y 502.661,Z 389.976,A -85,B 0,C 180,E1 -5746.25,E2 -5746.25} C_VEL
LIN {X 0,Y 502.713,Z 387.87,A -85,B 0,C 180,E1 -5747.895,E2 -5747.895} C_VEL
LIN {X 0,Y 502.835,Z 387.856,A -85,B 0,C 180,E1 -5750.345,E2 -5750.345} C_VEL
LIN {X 0,Y 502.932,Z 387.84,A -85,B 0,C 180,E1 -5752.814,E2 -5752.814} C_VEL
LIN {X 0,Y 502.868,Z 387.848,A -85,B 0,C 180,E1 -5755.19,E2 -5755.19} C_VEL
LIN {X 0,Y 503.021,Z 387.831,A -85,B 0,C 180,E1 -5757.598,E2 -5757.598} C_VEL
LIN {X 0,Y 503.022,Z 387.829,A -85,B 0,C 180,E1 -5760,E2 -5760} C_VEL
LIN {X 0,Y 503.02,Z 387.827,A -85,B 0,C 180,E1 -5762.402,E2 -5762.402} C_VEL
LIN {X 0,Y 502.935,Z 387.84,A -85,B 0,C 180,E1 -5765.614,E2 -5765.614} C_VEL
LIN {X 0,Y 502.898,Z 387.845,A -85,B 0,C 180,E1 -5768.033,E2 -5768.033} C_VEL
LIN {X 0,Y 502.873,Z 387.848,A -85,B 0,C 180,E1 -5771.283,E2 -5771.283} C_VEL
LIN {X 0,Y 502.841,Z 387.851,A -85,B 0,C 180,E1 -5774.571,E2 -5774.571} C_VEL
LIN {X 0,Y 502.858,Z 387.849,A -85,B 0,C 180,E1 -5777.907,E2 -5777.907} C_VEL
LIN {X 0,Y 502.825,Z 387.854,A -85,B 0,C 180,E1 -5780.537,E2 -5780.537} C_VEL
LIN {X 0,Y 502.793,Z 387.857,A -85,B 0,C 180,E1 -5783.041,E2 -5783.041} C_VEL
LIN {X 0,Y 502.838,Z 387.853,A -85,B 0,C 180,E1 -5785.676,E2 -5785.676} C_VEL
LIN {X 0,Y 502.839,Z 387.851,A -85,B 0,C 180,E1 -5788.373,E2 -5788.373} C_VEL
LIN {X 0,Y 502.791,Z 387.857,A -85,B 0,C 180,E1 -5791.5,E2 -5791.5} C_VEL
LIN {X 0,Y 502.802,Z 387.856,A -85,B 0,C 180,E1 -5794.445,E2 -5794.445} C_VEL
LIN {X 0,Y 502.779,Z 387.861,A -85,B 0,C 180,E1 -5797.179,E2 -5797.179} C_VEL
LIN {X 0,Y 502.824,Z 387.855,A -85,B 0,C 180,E1 -5800.012,E2 -5800.012} C_VEL
LIN {X 0,Y 502.772,Z 387.861,A -85,B 0,C 180,E1 -5803.232,E2 -5803.232} C_VEL
LIN {X 0,Y 502.788,Z 387.858,A -85,B 0,C 180,E1 -5805.662,E2 -5805.662} C_VEL
LIN {X 0,Y 502.826,Z 387.854,A -85,B 0,C 180,E1 -5809.005,E2 -5809.005} C_VEL
LIN {X 0,Y 502.825,Z 387.86,A -85,B 0,C 180,E1 -5811.373,E2 -5811.373} C_VEL
LIN {X 0,Y 503.684,Z 393.461,A -85,B 0,C 180,E1 -5814.027,E2 -5814.027} C_VEL
LIN {X 0,Y 503.653,Z 398.181,A -85,B 0,C 180,E1 -5816.072,E2 -5816.072} C_VEL
LIN {X 0,Y 503.321,Z 405.01,A -85,B 0,C 180,E1 -5818.893,E2 -5818.893} C_VEL
LIN {X 0,Y 503.089,Z 411.959,A -85,B 0,C 180,E1 -5821.654,E2 -5821.654} C_VEL
LIN {X 0,Y 502.849,Z 420.163,A -85,B 0,C 180,E1 -5824.769,E2 -5824.769} C_VEL
LIN {X 0,Y 502.685,Z 428.438,A -85,B 0,C 180,E1 -5827.823,E2 -5827.823} C_VEL
LIN {X 0,Y 502.515,Z 436.831,A -85,B 0,C 180,E1 -5830.813,E2 -5830.813} C_VEL
LIN {X 0,Y 502.394,Z 446.469,A -85,B 0,C 180,E1 -5834.17,E2 -5834.17} C_VEL
LIN {X 0,Y 502.34,Z 451.131,A -85,B 0,C 180,E1 -5835.712,E2 -5835.712} C_VEL
LIN {X 0,Y 504.416,Z 464.395,A -85,B 0,C 180,E1 -5836.094,E2 -5836.094} C_VEL
LIN {X 0,Y 504.344,Z 476.654,A -85,B 0,C 180,E1 -5836.554,E2 -5836.554} C_VEL
LIN {X 0,Y 503.941,Z 489.288,A -85,B 0,C 180,E1 -5837.194,E2 -5837.194} C_VEL
LIN {X 0,Y 503.605,Z 500.285,A -85,B 0,C 180,E1 -5837.917,E2 -5837.917} C_VEL
LIN {X 0,Y 503.268,Z 511.26,A -85,B 0,C 180,E1 -5838.828,E2 -5838.828} C_VEL
LIN {X 0,Y 502.959,Z 520.206,A -85,B 0,C 180,E1 -5839.738,E2 -5839.738} C_VEL
LIN {X 0,Y 502.657,Z 529.928,A -85,B 0,C 180,E1 -5840.951,E2 -5840.951} C_VEL
LIN {X 0,Y 502.413,Z 537.671,A -85,B 0,C 180,E1 -5842.161,E2 -5842.161} C_VEL
LIN {X 0,Y 502.236,Z 544.394,A -85,B 0,C 180,E1 -5843.482,E2 -5843.482} C_VEL
LIN {X 0,Y 502.177,Z 549.557,A -85,B 0,C 180,E1 -5844.781,E2 -5844.781} C_VEL
LIN {X 0,Y 502.145,Z 553.186,A -85,B 0,C 180,E1 -5845.988,E2 -5845.988} C_VEL
LIN {X 0,Y 502.121,Z 555.06,A -85,B 0,C 180,E1 -5846.791,E2 -5846.791} C_VEL
LIN {X 0,Y 502.092,Z 556.463,A -85,B 0,C 180,E1 -5847.594,E2 -5847.594} C_VEL
LIN {X 0,Y 501.99,Z 558.076,A -85,B 0,C 180,E1 -5849.198,E2 -5849.198} C_VEL
LIN {X 0,Y 501.98,Z 558.296,A -85,B 0,C 180,E1 -5850,E2 -5850} C_VEL
LIN {X 0,Y 502.036,Z 557.475,A -85,B 0,C 180,E1 -5851.605,E2 -5851.605} C_VEL
LIN {X 0,Y 502.092,Z 556.481,A -85,B 0,C 180,E1 -5852.407,E2 -5852.407} C_VEL
LIN {X 0,Y 502.121,Z 555.083,A -85,B 0,C 180,E1 -5853.21,E2 -5853.21} C_VEL
LIN {X 0,Y 502.112,Z 552.14,A -85,B 0,C 180,E1 -5854.415,E2 -5854.415} C_VEL
LIN {X 0,Y 502.225,Z 548.157,A -85,B 0,C 180,E1 -5855.622,E2 -5855.622} C_VEL
LIN {X 0,Y 502.333,Z 542.127,A -85,B 0,C 180,E1 -5857.012,E2 -5857.012} C_VEL
LIN {X 0,Y 502.495,Z 535.327,A -85,B 0,C 180,E1 -5858.242,E2 -5858.242} C_VEL
LIN {X 0,Y 502.755,Z 527.018,A -85,B 0,C 180,E1 -5859.454,E2 -5859.454} C_VEL
LIN {X 0,Y 502.997,Z 518.495,A -85,B 0,C 180,E1 -5860.465,E2 -5860.465} C_VEL
LIN {X 0,Y 503.42,Z 507.972,A -85,B 0,C 180,E1 -5861.475,E2 -5861.475} C_VEL
LIN {X 0,Y 503.696,Z 496.813,A -85,B 0,C 180,E1 -5862.339,E2 -5862.339} C_VEL
LIN {X 0,Y 504.05,Z 486.161,A -85,B 0,C 180,E1 -5862.993,E2 -5862.993} C_VEL
LIN {X 0,Y 504.392,Z 474.438,A -85,B 0,C 180,E1 -5863.548,E2 -5863.548} C_VEL
LIN {X 0,Y 504.451,Z 464.57,A -85,B 0,C 180,E1 -5863.906,E2 -5863.906} C_VEL
LIN {X 0,Y 502.41,Z 452.052,A -85,B 0,C 180,E1 -5864.274,E2 -5864.274} C_VEL
LIN {X 0,Y 502.322,Z 451.13,A -85,B 0,C 180,E1 -5864.302,E2 -5864.302} C_VEL
LIN {X 0,Y 502.45,Z 443.206,A -85,B 0,C 180,E1 -5867.082,E2 -5867.082} C_VEL
LIN {X 0,Y 502.608,Z 434.811,A -85,B 0,C 180,E1 -5870.035,E2 -5870.035} C_VEL
LIN {X 0,Y 502.758,Z 426.481,A -85,B 0,C 180,E1 -5873.042,E2 -5873.042} C_VEL
LIN {X 0,Y 502.972,Z 418.229,A -85,B 0,C 180,E1 -5876.113,E2 -5876.113} C_VEL
LIN {X 0,Y 503.202,Z 409.998,A -85,B 0,C 180,E1 -5879.264,E2 -5879.264} C_VEL
LIN {X 0,Y 503.455,Z 402.995,A -85,B 0,C 180,E1 -5882.037,E2 -5882.037} C_VEL
LIN {X 0,Y 503.78,Z 396.019,A -85,B 0,C 180,E1 -5884.888,E2 -5884.888} C_VEL
LIN {X 0,Y 503.435,Z 391.415,A -85,B 0,C 180,E1 -5886.89,E2 -5886.89} C_VEL
LIN {X 0,Y 502.812,Z 387.855,A -85,B 0,C 180,E1 -5888.558,E2 -5888.558} C_VEL
LIN {X 0,Y 502.822,Z 387.855,A -85,B 0,C 180,E1 -5891.066,E2 -5891.066} C_VEL
LIN {X 0,Y 502.787,Z 387.859,A -85,B 0,C 180,E1 -5894.53,E2 -5894.53} C_VEL
LIN {X 0,Y 502.796,Z 387.856,A -85,B 0,C 180,E1 -5897.86,E2 -5897.86} C_VEL
LIN {X 0,Y 502.802,Z 387.856,A -85,B 0,C 180,E1 -5901.024,E2 -5901.024} C_VEL
LIN {X 0,Y 502.783,Z 387.858,A -85,B 0,C 180,E1 -5904.168,E2 -5904.168} C_VEL
LIN {X 0,Y 502.831,Z 387.852,A -85,B 0,C 180,E1 -5906.994,E2 -5906.994} C_VEL
LIN {X 0,Y 502.816,Z 387.854,A -85,B 0,C 180,E1 -5910.065,E2 -5910.065} C_VEL
LIN {X 0,Y 502.833,Z 387.852,A -85,B 0,C 180,E1 -5912.533,E2 -5912.533} C_VEL
LIN {X 0,Y 502.827,Z 387.852,A -85,B 0,C 180,E1 -5915.299,E2 -5915.299} C_VEL
LIN {X 0,Y 502.781,Z 387.856,A -85,B 0,C 180,E1 -5917.826,E2 -5917.826} C_VEL
LIN {X 0,Y 502.825,Z 387.851,A -85,B 0,C 180,E1 -5920.4,E2 -5920.4} C_VEL
LIN {X 0,Y 502.83,Z 387.852,A -85,B 0,C 180,E1 -5922.931,E2 -5922.931} C_VEL
LIN {X 0,Y 502.845,Z 387.851,A -85,B 0,C 180,E1 -5925.429,E2 -5925.429} C_VEL
LIN {X 0,Y 502.877,Z 387.846,A -85,B 0,C 180,E1 -5928.717,E2 -5928.717} C_VEL
LIN {X 0,Y 502.902,Z 387.842,A -85,B 0,C 180,E1 -5931.967,E2 -5931.967} C_VEL
LIN {X 0,Y 502.938,Z 387.839,A -85,B 0,C 180,E1 -5934.386,E2 -5934.386} C_VEL
LIN {X 0,Y 503.023,Z 387.829,A -85,B 0,C 180,E1 -5937.598,E2 -5937.598} C_VEL
LIN {X 0,Y 503.028,Z 387.827,A -85,B 0,C 180,E1 -5940,E2 -5940} C_VEL
LIN {X 0,Y 503.023,Z 387.828,A -85,B 0,C 180,E1 -5942.402,E2 -5942.402} C_VEL
LIN {X 0,Y 502.928,Z 387.84,A -85,B 0,C 180,E1 -5946.419,E2 -5946.419} C_VEL
LIN {X 0,Y 502.874,Z 387.847,A -85,B 0,C 180,E1 -5948.843,E2 -5948.843} C_VEL
LIN {X 0,Y 502.846,Z 387.851,A -85,B 0,C 180,E1 -5952.102,E2 -5952.102} C_VEL
LIN {X 0,Y 502.849,Z 387.851,A -85,B 0,C 180,E1 -5955.4,E2 -5955.4} C_VEL
LIN {X 0,Y 502.847,Z 387.851,A -85,B 0,C 180,E1 -5958.122,E2 -5958.122} C_VEL
LIN {X 0,Y 502.829,Z 387.853,A -85,B 0,C 180,E1 -5960.536,E2 -5960.536} C_VEL
LIN {X 0,Y 502.791,Z 387.857,A -85,B 0,C 180,E1 -5963.041,E2 -5963.041} C_VEL
LIN {X 0,Y 502.84,Z 387.849,A -85,B 0,C 180,E1 -5965.676,E2 -5965.676} C_VEL
LIN {X 0,Y 502.84,Z 387.85,A -85,B 0,C 180,E1 -5968.373,E2 -5968.373} C_VEL
LIN {X 0,Y 502.794,Z 387.855,A -85,B 0,C 180,E1 -5971.499,E2 -5971.499} C_VEL
LIN {X 0,Y 502.806,Z 387.855,A -85,B 0,C 180,E1 -5974.444,E2 -5974.444} C_VEL
LIN {X 0,Y 502.782,Z 387.858,A -85,B 0,C 180,E1 -5977.178,E2 -5977.178} C_VEL
LIN {X 0,Y 502.788,Z 387.856,A -85,B 0,C 180,E1 -5980.015,E2 -5980.015} C_VEL
LIN {X 0,Y 502.804,Z 387.855,A -85,B 0,C 180,E1 -5982.199,E2 -5982.199} C_VEL
LIN {X 0,Y 502.786,Z 387.857,A -85,B 0,C 180,E1 -5985.47,E2 -5985.47} C_VEL
LIN {X 0,Y 502.822,Z 387.854,A -85,B 0,C 180,E1 -5988.934,E2 -5988.934} C_VEL
LIN {X 0,Y 502.794,Z 387.855,A -85,B 0,C 180,E1 -5992.046,E2 -5992.046} C_VEL
LIN {X 0,Y 502.809,Z 387.854,A -85,B 0,C 180,E1 -5995.035,E2 -5995.035} C_VEL
LIN {X 0,Y 502.81,Z 387.853,A -85,B 0,C 180,E1 -5997.218,E2 -5997.218} C_VEL
LIN {X 0,Y 502.108,Z 387.941,A -85,B 0,C 180,E1 -5997.887,E2 -5997.887} C_VEL
LIN {X 0,Y 499.243,Z 388.298,A -85,B 0,C 180,E1 -5998.972,E2 -5998.972} C_VEL
LIN {X 0,Y 496.849,Z 388.598,A -85,B 0,C 180,E1 -5999.847,E2 -5999.847} C_VEL
LIN {X 0,Y 495.833,Z 388.724,A -85,B 0,C 180,E1 -6000.523,E2 -6000.523} C_VEL
LIN {X 0,Y 495.755,Z 388.73,A -85,B 0,C 180,E1 -6000.752,E2 -6000.752} C_VEL
LIN {X 0,Y 495.793,Z 388.728,A -85,B 0,C 180,E1 -6003.932,E2 -6003.932} C_VEL
LIN {X 0,Y 495.762,Z 388.731,A -85,B 0,C 180,E1 -6007.139,E2 -6007.139} C_VEL
LIN {X 0,Y 495.774,Z 388.731,A -85,B 0,C 180,E1 -6010.11,E2 -6010.11} C_VEL
LIN {X 0,Y 495.783,Z 388.732,A -85,B 0,C 180,E1 -6012.681,E2 -6012.681} C_VEL
LIN {X 0,Y 495.792,Z 388.729,A -85,B 0,C 180,E1 -6015.217,E2 -6015.217} C_VEL
LIN {X 0,Y 495.854,Z 388.722,A -85,B 0,C 180,E1 -6018.555,E2 -6018.555} C_VEL
LIN {X 0,Y 495.875,Z 388.718,A -85,B 0,C 180,E1 -6021.852,E2 -6021.852} C_VEL
LIN {X 0,Y 495.898,Z 388.716,A -85,B 0,C 180,E1 -6024.306,E2 -6024.306} C_VEL
LIN {X 0,Y 495.996,Z 388.703,A -85,B 0,C 180,E1 -6027.563,E2 -6027.563} C_VEL
LIN {X 0,Y 495.985,Z 388.704,A -85,B 0,C 180,E1 -6030.812,E2 -6030.812} C_VEL
LIN {X 0,Y 495.996,Z 388.703,A -85,B 0,C 180,E1 -6032.436,E2 -6032.436} C_VEL
LIN {X 0,Y 495.884,Z 388.718,A -85,B 0,C 180,E1 -6035.693,E2 -6035.693} C_VEL
LIN {X 0,Y 495.703,Z 388.742,A -85,B 0,C 180,E1 -6038.15,E2 -6038.15} C_VEL
LIN {X 0,Y 495.602,Z 388.889,A -85,B 0,C 180,E1 -6038.974,E2 -6038.974} C_VEL
LIN {X 0,Y 495.518,Z 392.767,A -85,B 0,C 180,E1 -6041.864,E2 -6041.864} C_VEL
LIN {X 0,Y 495.385,Z 397.425,A -85,B 0,C 180,E1 -6045.266,E2 -6045.266} C_VEL
LIN {X 0,Y 495.284,Z 401.493,A -85,B 0,C 180,E1 -6048.19,E2 -6048.19} C_VEL
LIN {X 0,Y 495.174,Z 405.166,A -85,B 0,C 180,E1 -6050.782,E2 -6050.782} C_VEL
LIN {X 0,Y 495.13,Z 408.903,A -85,B 0,C 180,E1 -6053.418,E2 -6053.418} C_VEL
LIN {X 0,Y 495.041,Z 413.487,A -85,B 0,C 180,E1 -6056.569,E2 -6056.569} C_VEL
LIN {X 0,Y 495.027,Z 416.593,A -85,B 0,C 180,E1 -6058.59,E2 -6058.59} C_VEL
LIN {X 0,Y 497.484,Z 428.663,A -85,B 0,C 180,E1 -6058.995,E2 -6058.995} C_VEL
LIN {X 0,Y 497.713,Z 432.975,A -85,B 0,C 180,E1 -6059.153,E2 -6059.153} C_VEL
LIN {X 0,Y 497.309,Z 445.361,A -85,B 0,C 180,E1 -6059.701,E2 -6059.701} C_VEL
LIN {X 0,Y 496.931,Z 456.893,A -85,B 0,C 180,E1 -6060.377,E2 -6060.377} C_VEL
LIN {X 0,Y 496.6,Z 468.12,A -85,B 0,C 180,E1 -6061.219,E2 -6061.219} C_VEL
LIN {X 0,Y 496.237,Z 478.829,A -85,B 0,C 180,E1 -6062.234,E2 -6062.234} C_VEL
LIN {X 0,Y 495.91,Z 488.549,A -85,B 0,C 180,E1 -6063.375,E2 -6063.375} C_VEL
LIN {X 0,Y 495.556,Z 497.232,A -85,B 0,C 180,E1 -6064.658,E2 -6064.658} C_VEL
LIN {X 0,Y 495.313,Z 504.571,A -85,B 0,C 180,E1 -6066.024,E2 -6066.024} C_VEL
LIN {X 0,Y 495.148,Z 510.145,A -85,B 0,C 180,E1 -6067.359,E2 -6067.359} C_VEL
LIN {X 0,Y 495.065,Z 514.285,A -85,B 0,C 180,E1 -6068.667,E2 -6068.667} C_VEL
LIN {X 0,Y 494.967,Z 517.202,A -85,B 0,C 180,E1 -6069.938,E2 -6069.938} C_VEL
LIN {X 0,Y 494.874,Z 519.067,A -85,B 0,C 180,E1 -6071.176,E2 -6071.176} C_VEL
LIN {X 0,Y 494.902,Z 519.997,A -85,B 0,C 180,E1 -6072.401,E2 -6072.401} C_VEL
LIN {X 0,Y 494.938,Z 519.778,A -85,B 0,C 180,E1 -6074.089,E2 -6074.089} C_VEL
LIN {X 0,Y 494.945,Z 518.684,A -85,B 0,C 180,E1 -6075.232,E2 -6075.232} C_VEL
LIN {X 0,Y 495.015,Z 516.772,A -85,B 0,C 180,E1 -6076.391,E2 -6076.391} C_VEL
LIN {X 0,Y 495.09,Z 513.932,A -85,B 0,C 180,E1 -6077.574,E2 -6077.574} C_VEL
LIN {X 0,Y 495.15,Z 510.015,A -85,B 0,C 180,E1 -6078.786,E2 -6078.786} C_VEL
LIN {X 0,Y 495.307,Z 504.902,A -85,B 0,C 180,E1 -6080.014,E2 -6080.014} C_VEL
LIN {X 0,Y 495.571,Z 497.565,A -85,B 0,C 180,E1 -6081.392,E2 -6081.392} C_VEL
LIN {X 0,Y 495.799,Z 489.942,A -85,B 0,C 180,E1 -6082.541,E2 -6082.541} C_VEL
LIN {X 0,Y 496.17,Z 480.496,A -85,B 0,C 180,E1 -6083.694,E2 -6083.694} C_VEL
LIN {X 0,Y 496.6,Z 470.012,A -85,B 0,C 180,E1 -6084.715,E2 -6084.715} C_VEL
LIN {X 0,Y 496.959,Z 459.387,A -85,B 0,C 180,E1 -6085.55,E2 -6085.55} C_VEL
LIN {X 0,Y 497.296,Z 448.448,A -85,B 0,C 180,E1 -6086.235,E2 -6086.235} C_VEL
LIN {X 0,Y 497.65,Z 435.609,A -85,B 0,C 180,E1 -6086.839,E2 -6086.839} C_VEL
LIN {X 0,Y 497.526,Z 428.819,A -85,B 0,C 180,E1 -6087.095,E2 -6087.095} C_VEL
LIN {X 0,Y 495.47,Z 418.59,A -85,B 0,C 180,E1 -6087.444,E2 -6087.444} C_VEL
LIN {X 0,Y 495.065,Z 416.693,A -85,B 0,C 180,E1 -6087.504,E2 -6087.504} C_VEL
LIN {X 0,Y 495.131,Z 412.802,A -85,B 0,C 180,E1 -6090.212,E2 -6090.212} C_VEL
LIN {X 0,Y 495.22,Z 408.316,A -85,B 0,C 180,E1 -6093.388,E2 -6093.388} C_VEL
LIN {X 0,Y 495.284,Z 405.105,A -85,B 0,C 180,E1 -6095.701,E2 -6095.701} C_VEL
LIN {X 0,Y 495.373,Z 401.451,A -85,B 0,C 180,E1 -6098.354,E2 -6098.354} C_VEL
LIN {X 0,Y 495.461,Z 397.925,A -85,B 0,C 180,E1 -6100.959,E2 -6100.959} C_VEL
LIN {X 0,Y 495.508,Z 394.479,A -85,B 0,C 180,E1 -6103.521,E2 -6103.521} C_VEL
LIN {X 0,Y 495.599,Z 391.129,A -85,B 0,C 180,E1 -6106.05,E2 -6106.05} C_VEL
LIN {X 0,Y 495.701,Z 388.743,A -85,B 0,C 180,E1 -6108.032,E2 -6108.032} C_VEL
LIN {X 0,Y 495.84,Z 388.726,A -85,B 0,C 180,E1 -6111.03,E2 -6111.03} C_VEL
LIN {X 0,Y 495.875,Z 388.72,A -85,B 0,C 180,E1 -6113.49,E2 -6113.49} C_VEL
LIN {X 0,Y 495.843,Z 388.724,A -85,B 0,C 180,E1 -6116.75,E2 -6116.75} C_VEL
LIN {X 0,Y 496.003,Z 388.703,A -85,B 0,C 180,E1 -6119.188,E2 -6119.188} C_VEL
LIN {X 0,Y 495.867,Z 388.721,A -85,B 0,C 180,E1 -6121.624,E2 -6121.624} C_VEL
LIN {X 0,Y 495.84,Z 388.723,A -85,B 0,C 180,E1 -6123.25,E2 -6123.25} C_VEL
LIN {X 0,Y 495.876,Z 388.718,A -85,B 0,C 180,E1 -6126.51,E2 -6126.51} C_VEL
LIN {X 0,Y 495.839,Z 388.725,A -85,B 0,C 180,E1 -6128.97,E2 -6128.97} C_VEL
LIN {X 0,Y 495.824,Z 388.726,A -85,B 0,C 180,E1 -6132.035,E2 -6132.035} C_VEL
LIN {X 0,Y 495.82,Z 388.726,A -85,B 0,C 180,E1 -6135.452,E2 -6135.452} C_VEL
LIN {X 0,Y 495.802,Z 388.729,A -85,B 0,C 180,E1 -6138.248,E2 -6138.248} C_VEL
LIN {X 0,Y 495.77,Z 388.732,A -85,B 0,C 180,E1 -6140.757,E2 -6140.757} C_VEL
LIN {X 0,Y 495.749,Z 388.735,A -85,B 0,C 180,E1 -6143.387,E2 -6143.387} C_VEL
LIN {X 0,Y 495.796,Z 388.728,A -85,B 0,C 180,E1 -6146.068,E2 -6146.068} C_VEL
LIN {X 0,Y 495.778,Z 388.733,A -85,B 0,C 180,E1 -6148.815,E2 -6148.815} C_VEL
LIN {X 0,Y 495.754,Z 388.734,A -85,B 0,C 180,E1 -6151.726,E2 -6151.726} C_VEL
LIN {X 0,Y 495.772,Z 388.732,A -85,B 0,C 180,E1 -6154.696,E2 -6154.696} C_VEL
LIN {X 0,Y 495.73,Z 388.738,A -85,B 0,C 180,E1 -6157.562,E2 -6157.562} C_VEL
LIN {X 0,Y 495.791,Z 388.731,A -85,B 0,C 180,E1 -6160.052,E2 -6160.052} C_VEL
LIN {X 0,Y 495.724,Z 388.738,A -85,B 0,C 180,E1 -6162.884,E2 -6162.884} C_VEL
LIN {X 0,Y 495.732,Z 388.736,A -85,B 0,C 180,E1 -6166,E2 -6166} C_VEL
LIN {X 0,Y 495.779,Z 388.732,A -85,B 0,C 180,E1 -6169.302,E2 -6169.302} C_VEL
LIN {X 0,Y 495.814,Z 388.931,A -85,B 0,C 180,E1 -6171.225,E2 -6171.225} C_VEL
LIN {X 0,Y 496.651,Z 394.185,A -85,B 0,C 180,E1 -6173.765,E2 -6173.765} C_VEL
LIN {X 0,Y 496.665,Z 399.258,A -85,B 0,C 180,E1 -6176.018,E2 -6176.018} C_VEL
LIN {X 0,Y 496.297,Z 406.033,A -85,B 0,C 180,E1 -6178.878,E2 -6178.878} C_VEL
LIN {X 0,Y 496.064,Z 412.407,A -85,B 0,C 180,E1 -6181.449,E2 -6181.449} C_VEL
LIN {X 0,Y 495.844,Z 419.985,A -85,B 0,C 180,E1 -6184.387,E2 -6184.387} C_VEL
LIN {X 0,Y 495.653,Z 428.242,A -85,B 0,C 180,E1 -6187.491,E2 -6187.491} C_VEL
LIN {X 0,Y 495.457,Z 436.579,A -85,B 0,C 180,E1 -6190.529,E2 -6190.529} C_VEL
LIN {X 0,Y 495.329,Z 444.961,A -85,B 0,C 180,E1 -6193.515,E2 -6193.515} C_VEL
LIN {X 0,Y 495.242,Z 450.589,A -85,B 0,C 180,E1 -6195.49,E2 -6195.49} C_VEL
LIN {X 0,Y 497.407,Z 464.815,A -85,B 0,C 180,E1 -6195.92,E2 -6195.92} C_VEL
LIN {X 0,Y 497.605,Z 468.616,A -85,B 0,C 180,E1 -6196.056,E2 -6196.056} C_VEL
LIN {X 0,Y 497.274,Z 480.738,A -85,B 0,C 180,E1 -6196.567,E2 -6196.567} C_VEL
LIN {X 0,Y 496.889,Z 492.192,A -85,B 0,C 180,E1 -6197.212,E2 -6197.212} C_VEL
LIN {X 0,Y 496.51,Z 503.881,A -85,B 0,C 180,E1 -6198.053,E2 -6198.053} C_VEL
LIN {X 0,Y 496.183,Z 514.15,A -85,B 0,C 180,E1 -6198.977,E2 -6198.977} C_VEL
LIN {X 0,Y 495.817,Z 523.381,A -85,B 0,C 180,E1 -6200.001,E2 -6200.001} C_VEL
LIN {X 0,Y 495.51,Z 532.378,A -85,B 0,C 180,E1 -6201.23,E2 -6201.23} C_VEL
LIN {X 0,Y 495.286,Z 539.625,A -85,B 0,C 180,E1 -6202.458,E2 -6202.458} C_VEL
LIN {X 0,Y 495.137,Z 545.652,A -85,B 0,C 180,E1 -6203.746,E2 -6203.746} C_VEL
LIN {X 0,Y 495.037,Z 550.59,A -85,B 0,C 180,E1 -6205.114,E2 -6205.114} C_VEL
LIN {X 0,Y 495.04,Z 552.904,A -85,B 0,C 180,E1 -6205.93,E2 -6205.93} C_VEL
LIN {X 0,Y 495.042,Z 554.782,A -85,B 0,C 180,E1 -6206.745,E2 -6206.745} C_VEL
LIN {X 0,Y 494.998,Z 556.187,A -85,B 0,C 180,E1 -6207.559,E2 -6207.559} C_VEL
LIN {X 0,Y 494.962,Z 557.189,A -85,B 0,C 180,E1 -6208.373,E2 -6208.373} C_VEL
LIN {X 0,Y 494.898,Z 558.025,A -85,B 0,C 180,E1 -6210,E2 -6210} C_VEL
LIN {X 0,Y 494.962,Z 557.206,A -85,B 0,C 180,E1 -6211.628,E2 -6211.628} C_VEL
LIN {X 0,Y 494.998,Z 556.211,A -85,B 0,C 180,E1 -6212.441,E2 -6212.441} C_VEL
LIN {X 0,Y 495.042,Z 554.813,A -85,B 0,C 180,E1 -6213.256,E2 -6213.256} C_VEL
LIN {X 0,Y 495.016,Z 551.868,A -85,B 0,C 180,E1 -6214.479,E2 -6214.479} C_VEL
LIN {X 0,Y 495.143,Z 547.884,A -85,B 0,C 180,E1 -6215.702,E2 -6215.702} C_VEL
LIN {X 0,Y 495.257,Z 541.749,A -85,B 0,C 180,E1 -6217.133,E2 -6217.133} C_VEL
LIN {X 0,Y 495.442,Z 535.048,A -85,B 0,C 180,E1 -6218.361,E2 -6218.361} C_VEL
LIN {X 0,Y 495.724,Z 526.736,A -85,B 0,C 180,E1 -6219.589,E2 -6219.589} C_VEL
LIN {X 0,Y 495.993,Z 518.208,A -85,B 0,C 180,E1 -6220.615,E2 -6220.615} C_VEL
LIN {X 0,Y 496.445,Z 507.681,A -85,B 0,C 180,E1 -6221.639,E2 -6221.639} C_VEL
LIN {X 0,Y 496.745,Z 496.456,A -85,B 0,C 180,E1 -6222.519,E2 -6222.519} C_VEL
LIN {X 0,Y 497.101,Z 485.861,A -85,B 0,C 180,E1 -6223.178,E2 -6223.178} C_VEL
LIN {X 0,Y 497.474,Z 474.129,A -85,B 0,C 180,E1 -6223.74,E2 -6223.74} C_VEL
LIN {X 0,Y 497.511,Z 465.413,A -85,B 0,C 180,E1 -6224.065,E2 -6224.065} C_VEL
LIN {X 0,Y 495.468,Z 452.477,A -85,B 0,C 180,E1 -6224.465,E2 -6224.465} C_VEL
LIN {X 0,Y 495.233,Z 450.796,A -85,B 0,C 180,E1 -6224.537,E2 -6224.537} C_VEL
LIN {X 0,Y 495.371,Z 442.942,A -85,B 0,C 180,E1 -6227.334,E2 -6227.334} C_VEL
LIN {X 0,Y 495.525,Z 435.792,A -85,B 0,C 180,E1 -6229.901,E2 -6229.901} C_VEL
LIN {X 0,Y 495.686,Z 427.802,A -85,B 0,C 180,E1 -6232.84,E2 -6232.84} C_VEL
LIN {X 0,Y 495.913,Z 419.249,A -85,B 0,C 180,E1 -6236.061,E2 -6236.061} C_VEL
LIN {X 0,Y 496.184,Z 411.04,A -85,B 0,C 180,E1 -6239.253,E2 -6239.253} C_VEL
LIN {X 0,Y 496.421,Z 404.571,A -85,B 0,C 180,E1 -6241.849,E2 -6241.849} C_VEL
LIN {X 0,Y 496.773,Z 397.315,A -85,B 0,C 180,E1 -6244.86,E2 -6244.86} C_VEL
LIN {X 0,Y 496.431,Z 392.469,A -85,B 0,C 180,E1 -6246.99,E2 -6246.99} C_VEL
LIN {X 0,Y 495.775,Z 388.732,A -85,B 0,C 180,E1 -6248.769,E2 -6248.769} C_VEL
LIN {X 0,Y 495.759,Z 388.733,A -85,B 0,C 180,E1 -6251.781,E2 -6251.781} C_VEL
LIN {X 0,Y 495.738,Z 388.736,A -85,B 0,C 180,E1 -6255.141,E2 -6255.141} C_VEL
LIN {X 0,Y 495.757,Z 388.733,A -85,B 0,C 180,E1 -6258.219,E2 -6258.219} C_VEL
LIN {X 0,Y 495.751,Z 388.734,A -85,B 0,C 180,E1 -6261.408,E2 -6261.408} C_VEL
LIN {X 0,Y 495.754,Z 388.734,A -85,B 0,C 180,E1 -6264.463,E2 -6264.463} C_VEL
LIN {X 0,Y 495.767,Z 388.732,A -85,B 0,C 180,E1 -6267.405,E2 -6267.405} C_VEL
LIN {X 0,Y 495.767,Z 388.732,A -85,B 0,C 180,E1 -6270.254,E2 -6270.254} C_VEL
LIN {X 0,Y 495.824,Z 388.725,A -85,B 0,C 180,E1 -6273.251,E2 -6273.251} C_VEL
LIN {X 0,Y 495.749,Z 388.734,A -85,B 0,C 180,E1 -6275.725,E2 -6275.725} C_VEL
LIN {X 0,Y 495.743,Z 388.734,A -85,B 0,C 180,E1 -6278.371,E2 -6278.371} C_VEL
LIN {X 0,Y 495.784,Z 388.732,A -85,B 0,C 180,E1 -6280.971,E2 -6280.971} C_VEL
LIN {X 0,Y 495.778,Z 388.73,A -85,B 0,C 180,E1 -6283.53,E2 -6283.53} C_VEL
LIN {X 0,Y 495.793,Z 388.728,A -85,B 0,C 180,E1 -6286.056,E2 -6286.056} C_VEL
LIN {X 0,Y 495.852,Z 388.721,A -85,B 0,C 180,E1 -6288.555,E2 -6288.555} C_VEL
LIN {X 0,Y 495.874,Z 388.718,A -85,B 0,C 180,E1 -6291.852,E2 -6291.852} C_VEL
LIN {X 0,Y 495.896,Z 388.717,A -85,B 0,C 180,E1 -6294.306,E2 -6294.306} C_VEL
LIN {X 0,Y 495.992,Z 388.704,A -85,B 0,C 180,E1 -6297.564,E2 -6297.564} C_VEL
LIN {X 0,Y 496.005,Z 388.702,A -85,B 0,C 180,E1 -6300.812,E2 -6300.812} C_VEL
LIN {X 0,Y 495.843,Z 388.723,A -85,B 0,C 180,E1 -6303.25,E2 -6303.25} C_VEL
LIN {X 0,Y 495.88,Z 388.718,A -85,B 0,C 180,E1 -6306.51,E2 -6306.51} C_VEL
LIN {X 0,Y 495.843,Z 388.722,A -85,B 0,C 180,E1 -6308.97,E2 -6308.97} C_VEL
LIN {X 0,Y 495.828,Z 388.724,A -85,B 0,C 180,E1 -6312.035,E2 -6312.035} C_VEL
LIN {X 0,Y 495.824,Z 388.725,A -85,B 0,C 180,E1 -6315.452,E2 -6315.452} C_VEL
LIN {X 0,Y 495.807,Z 388.727,A -85,B 0,C 180,E1 -6318.247,E2 -6318.247} C_VEL
LIN {X 0,Y 495.774,Z 388.731,A -85,B 0,C 180,E1 -6320.756,E2 -6320.756} C_VEL
LIN {X 0,Y 495.748,Z 388.733,A -85,B 0,C 180,E1 -6323.387,E2 -6323.387} C_VEL
LIN {X 0,Y 495.791,Z 388.728,A -85,B 0,C 180,E1 -6326.068,E2 -6326.068} C_VEL
LIN {X 0,Y 495.772,Z 388.732,A -85,B 0,C 180,E1 -6328.815,E2 -6328.815} C_VEL
LIN {X 0,Y 495.756,Z 388.731,A -85,B 0,C 180,E1 -6331.725,E2 -6331.725} C_VEL
LIN {X 0,Y 495.776,Z 388.733,A -85,B 0,C 180,E1 -6334.695,E2 -6334.695} C_VEL
LIN {X 0,Y 495.732,Z 388.734,A -85,B 0,C 180,E1 -6337.562,E2 -6337.562} C_VEL
LIN {X 0,Y 495.767,Z 388.733,A -85,B 0,C 180,E1 -6340.7,E2 -6340.7} C_VEL
LIN {X 0,Y 495.729,Z 388.736,A -85,B 0,C 180,E1 -6344.002,E2 -6344.002} C_VEL
LIN {X 0,Y 495.727,Z 388.736,A -85,B 0,C 180,E1 -6347.117,E2 -6347.117} C_VEL
LIN {X 0,Y 495.76,Z 388.732,A -85,B 0,C 180,E1 -6349.953,E2 -6349.953} C_VEL
LIN {X 0,Y 495.731,Z 388.738,A -85,B 0,C 180,E1 -6352.553,E2 -6352.553} C_VEL
LIN {X 0,Y 495.785,Z 388.727,A -85,B 0,C 180,E1 -6355.457,E2 -6355.457} C_VEL
LIN {X 0,Y 495.757,Z 388.734,A -85,B 0,C 180,E1 -6358.364,E2 -6358.364} C_VEL
LIN {X 0,Y 495.755,Z 388.73,A -85,B 0,C 180,E1 -6360.752,E2 -6360.752} C_VEL
LIN {X 0,Y 495.097,Z 388.814,A -85,B 0,C 180,E1 -6361.431,E2 -6361.431} C_VEL
LIN {X 0,Y 492.241,Z 389.171,A -85,B 0,C 180,E1 -6362.533,E2 -6362.533} C_VEL
LIN {X 0,Y 489.833,Z 389.47,A -85,B 0,C 180,E1 -6363.422,E2 -6363.422} C_VEL
LIN {X 0,Y 488.817,Z 389.597,A -85,B 0,C 180,E1 -6364.108,E2 -6364.108} C_VEL
LIN {X 0,Y 488.744,Z 389.608,A -85,B 0,C 180,E1 -6364.341,E2 -6364.341} C_VEL
LIN {X 0,Y 488.725,Z 389.607,A -85,B 0,C 180,E1 -6367.153,E2 -6367.153} C_VEL
LIN {X 0,Y 488.727,Z 389.608,A -85,B 0,C 180,E1 -6369.81,E2 -6369.81} C_VEL
LIN {X 0,Y 488.731,Z 389.608,A -85,B 0,C 180,E1 -6372.423,E2 -6372.423} C_VEL
LIN {X 0,Y 488.764,Z 389.605,A -85,B 0,C 180,E1 -6375,E2 -6375} C_VEL
LIN {X 0,Y 488.808,Z 389.599,A -85,B 0,C 180,E1 -6378.387,E2 -6378.387} C_VEL
LIN {X 0,Y 488.818,Z 389.596,A -85,B 0,C 180,E1 -6381.733,E2 -6381.733} C_VEL
LIN {X 0,Y 488.858,Z 389.592,A -85,B 0,C 180,E1 -6384.224,E2 -6384.224} C_VEL
LIN {X 0,Y 488.963,Z 389.579,A -85,B 0,C 180,E1 -6387.528,E2 -6387.528} C_VEL
LIN {X 0,Y 488.936,Z 389.582,A -85,B 0,C 180,E1 -6390.823,E2 -6390.823} C_VEL
LIN {X 0,Y 488.963,Z 389.579,A -85,B 0,C 180,E1 -6392.471,E2 -6392.471} C_VEL
LIN {X 0,Y 488.84,Z 389.595,A -85,B 0,C 180,E1 -6395.776,E2 -6395.776} C_VEL
LIN {X 0,Y 488.652,Z 389.62,A -85,B 0,C 180,E1 -6398.269,E2 -6398.269} C_VEL
LIN {X 0,Y 488.531,Z 389.869,A -85,B 0,C 180,E1 -6399.105,E2 -6399.105} C_VEL
LIN {X 0,Y 488.455,Z 393.619,A -85,B 0,C 180,E1 -6401.93,E2 -6401.93} C_VEL
LIN {X 0,Y 488.332,Z 398.27,A -85,B 0,C 180,E1 -6405.365,E2 -6405.365} C_VEL
LIN {X 0,Y 488.213,Z 402.546,A -85,B 0,C 180,E1 -6408.463,E2 -6408.463} C_VEL
LIN {X 0,Y 488.092,Z 406.241,A -85,B 0,C 180,E1 -6411.098,E2 -6411.098} C_VEL
LIN {X 0,Y 488.047,Z 410.018,A -85,B 0,C 180,E1 -6413.778,E2 -6413.778} C_VEL
LIN {X 0,Y 487.969,Z 414.293,A -85,B 0,C 180,E1 -6416.752,E2 -6416.752} C_VEL
LIN {X 0,Y 487.977,Z 416.797,A -85,B 0,C 180,E1 -6418.377,E2 -6418.377} C_VEL
LIN {X 0,Y 490.654,Z 429.934,A -85,B 0,C 180,E1 -6418.833,E2 -6418.833} C_VEL
LIN {X 0,Y 490.679,Z 439.131,A -85,B 0,C 180,E1 -6419.201,E2 -6419.201} C_VEL
LIN {X 0,Y 490.204,Z 451.19,A -85,B 0,C 180,E1 -6419.822,E2 -6419.822} C_VEL
LIN {X 0,Y 489.855,Z 462.628,A -85,B 0,C 180,E1 -6420.59,E2 -6420.59} C_VEL
LIN {X 0,Y 489.469,Z 473.191,A -85,B 0,C 180,E1 -6421.485,E2 -6421.485} C_VEL
LIN {X 0,Y 489.081,Z 483.754,A -85,B 0,C 180,E1 -6422.606,E2 -6422.606} C_VEL
LIN {X 0,Y 488.716,Z 492.659,A -85,B 0,C 180,E1 -6423.776,E2 -6423.776} C_VEL
LIN {X 0,Y 488.464,Z 499.623,A -85,B 0,C 180,E1 -6424.904,E2 -6424.904} C_VEL
LIN {X 0,Y 488.235,Z 506.43,A -85,B 0,C 180,E1 -6426.283,E2 -6426.283} C_VEL
LIN {X 0,Y 488.052,Z 511.603,A -85,B 0,C 180,E1 -6427.627,E2 -6427.627} C_VEL
LIN {X 0,Y 487.947,Z 515.42,A -85,B 0,C 180,E1 -6428.943,E2 -6428.943} C_VEL
LIN {X 0,Y 487.84,Z 518.368,A -85,B 0,C 180,E1 -6430.412,E2 -6430.412} C_VEL
LIN {X 0,Y 487.782,Z 519.686,A -85,B 0,C 180,E1 -6431.511,E2 -6431.511} C_VEL
LIN {X 0,Y 487.831,Z 520.334,A -85,B 0,C 180,E1 -6432.715,E2 -6432.715} C_VEL
LIN {X 0,Y 487.838,Z 520.157,A -85,B 0,C 180,E1 -6433.919,E2 -6433.919} C_VEL
LIN {X 0,Y 487.861,Z 519.18,A -85,B 0,C 180,E1 -6435.099,E2 -6435.099} C_VEL
LIN {X 0,Y 487.927,Z 517.394,A -85,B 0,C 180,E1 -6436.26,E2 -6436.26} C_VEL
LIN {X 0,Y 487.982,Z 514.83,A -85,B 0,C 180,E1 -6437.398,E2 -6437.398} C_VEL
LIN {X 0,Y 488.064,Z 511.489,A -85,B 0,C 180,E1 -6438.518,E2 -6438.518} C_VEL
LIN {X 0,Y 488.222,Z 505.8,A -85,B 0,C 180,E1 -6439.974,E2 -6439.974} C_VEL
LIN {X 0,Y 488.446,Z 499.729,A -85,B 0,C 180,E1 -6441.187,E2 -6441.187} C_VEL
LIN {X 0,Y 488.75,Z 492.033,A -85,B 0,C 180,E1 -6442.421,E2 -6442.421} C_VEL
LIN {X 0,Y 489.106,Z 483.105,A -85,B 0,C 180,E1 -6443.577,E2 -6443.577} C_VEL
LIN {X 0,Y 489.478,Z 473.701,A -85,B 0,C 180,E1 -6444.57,E2 -6444.57} C_VEL
LIN {X 0,Y 489.93,Z 462.968,A -85,B 0,C 180,E1 -6445.485,E2 -6445.485} C_VEL
LIN {X 0,Y 490.257,Z 451.708,A -85,B 0,C 180,E1 -6446.247,E2 -6446.247} C_VEL
LIN {X 0,Y 490.684,Z 439.055,A -85,B 0,C 180,E1 -6446.903,E2 -6446.903} C_VEL
LIN {X 0,Y 490.667,Z 429.833,A -85,B 0,C 180,E1 -6447.268,E2 -6447.268} C_VEL
LIN {X 0,Y 488.276,Z 418.544,A -85,B 0,C 180,E1 -6447.669,E2 -6447.669} C_VEL
LIN {X 0,Y 488.013,Z 416.949,A -85,B 0,C 180,E1 -6447.741,E2 -6447.741} C_VEL
LIN {X 0,Y 488.056,Z 412.772,A -85,B 0,C 180,E1 -6450.686,E2 -6450.686} C_VEL
LIN {X 0,Y 488.17,Z 408.857,A -85,B 0,C 180,E1 -6453.494,E2 -6453.494} C_VEL
LIN {X 0,Y 488.235,Z 405.109,A -85,B 0,C 180,E1 -6456.231,E2 -6456.231} C_VEL
LIN {X 0,Y 488.364,Z 400.938,A -85,B 0,C 180,E1 -6459.292,E2 -6459.292} C_VEL
LIN {X 0,Y 488.455,Z 396.773,A -85,B 0,C 180,E1 -6462.413,E2 -6462.413} C_VEL
LIN {X 0,Y 488.555,Z 393.385,A -85,B 0,C 180,E1 -6464.993,E2 -6464.993} C_VEL
LIN {X 0,Y 488.655,Z 389.621,A -85,B 0,C 180,E1 -6467.956,E2 -6467.956} C_VEL
LIN {X 0,Y 488.78,Z 389.605,A -85,B 0,C 180,E1 -6470.9,E2 -6470.9} C_VEL
LIN {X 0,Y 488.831,Z 389.598,A -85,B 0,C 180,E1 -6473.395,E2 -6473.395} C_VEL
LIN {X 0,Y 488.698,Z 389.613,A -85,B 0,C 180,E1 -6475.877,E2 -6475.877} C_VEL
LIN {X 0,Y 488.957,Z 389.582,A -85,B 0,C 180,E1 -6477.529,E2 -6477.529} C_VEL
LIN {X 0,Y 488.965,Z 389.58,A -85,B 0,C 180,E1 -6480,E2 -6480} C_VEL
LIN {X 0,Y 488.957,Z 389.579,A -85,B 0,C 180,E1 -6482.471,E2 -6482.471} C_VEL
LIN {X 0,Y 488.852,Z 389.595,A -85,B 0,C 180,E1 -6485.776,E2 -6485.776} C_VEL
LIN {X 0,Y 488.813,Z 389.599,A -85,B 0,C 180,E1 -6488.267,E2 -6488.267} C_VEL
LIN {X 0,Y 488.801,Z 389.6,A -85,B 0,C 180,E1 -6491.613,E2 -6491.613} C_VEL
LIN {X 0,Y 488.758,Z 389.605,A -85,B 0,C 180,E1 -6495.001,E2 -6495.001} C_VEL
LIN {X 0,Y 488.751,Z 389.607,A -85,B 0,C 180,E1 -6498.442,E2 -6498.442} C_VEL
LIN {X 0,Y 488.704,Z 389.611,A -85,B 0,C 180,E1 -6501.071,E2 -6501.071} C_VEL
LIN {X 0,Y 488.69,Z 389.613,A -85,B 0,C 180,E1 -6503.746,E2 -6503.746} C_VEL
LIN {X 0,Y 488.796,Z 389.601,A -85,B 0,C 180,E1 -6506.946,E2 -6506.946} C_VEL
LIN {X 0,Y 488.715,Z 389.61,A -85,B 0,C 180,E1 -6510.365,E2 -6510.365} C_VEL
LIN {X 0,Y 488.732,Z 389.608,A -85,B 0,C 180,E1 -6513.485,E2 -6513.485} C_VEL
LIN {X 0,Y 488.686,Z 389.616,A -85,B 0,C 180,E1 -6516.356,E2 -6516.356} C_VEL
LIN {X 0,Y 488.747,Z 389.61,A -85,B 0,C 180,E1 -6519.25,E2 -6519.25} C_VEL
LIN {X 0,Y 488.69,Z 389.615,A -85,B 0,C 180,E1 -6522.526,E2 -6522.526} C_VEL
LIN {X 0,Y 488.71,Z 389.612,A -85,B 0,C 180,E1 -6525.199,E2 -6525.199} C_VEL
LIN {X 0,Y 488.711,Z 389.608,A -85,B 0,C 180,E1 -6528.4,E2 -6528.4} C_VEL
LIN {X 0,Y 488.76,Z 389.739,A -85,B 0,C 180,E1 -6530.94,E2 -6530.94} C_VEL
LIN {X 0,Y 489.599,Z 394.914,A -85,B 0,C 180,E1 -6533.5,E2 -6533.5} C_VEL
LIN {X 0,Y 489.725,Z 399.191,A -85,B 0,C 180,E1 -6535.469,E2 -6535.469} C_VEL
LIN {X 0,Y 489.37,Z 405.969,A -85,B 0,C 180,E1 -6538.387,E2 -6538.387} C_VEL
LIN {X 0,Y 489.063,Z 412.856,A -85,B 0,C 180,E1 -6541.234,E2 -6541.234} C_VEL
LIN {X 0,Y 488.8,Z 420.973,A -85,B 0,C 180,E1 -6544.448,E2 -6544.448} C_VEL
LIN {X 0,Y 488.594,Z 429.237,A -85,B 0,C 180,E1 -6547.594,E2 -6547.594} C_VEL
LIN {X 0,Y 488.373,Z 437.528,A -85,B 0,C 180,E1 -6550.672,E2 -6550.672} C_VEL
LIN {X 0,Y 488.25,Z 445.879,A -85,B 0,C 180,E1 -6553.699,E2 -6553.699} C_VEL
LIN {X 0,Y 488.174,Z 450.414,A -85,B 0,C 180,E1 -6555.288,E2 -6555.288} C_VEL
LIN {X 0,Y 490.23,Z 464.066,A -85,B 0,C 180,E1 -6555.696,E2 -6555.696} C_VEL
LIN {X 0,Y 490.709,Z 468.258,A -85,B 0,C 180,E1 -6555.856,E2 -6555.856} C_VEL
LIN {X 0,Y 490.358,Z 480.396,A -85,B 0,C 180,E1 -6556.374,E2 -6556.374} C_VEL
LIN {X 0,Y 489.921,Z 492.648,A -85,B 0,C 180,E1 -6557.08,E2 -6557.08} C_VEL
LIN {X 0,Y 489.537,Z 503.552,A -85,B 0,C 180,E1 -6557.88,E2 -6557.88} C_VEL
LIN {X 0,Y 489.187,Z 513.83,A -85,B 0,C 180,E1 -6558.817,E2 -6558.817} C_VEL
LIN {X 0,Y 488.773,Z 523.069,A -85,B 0,C 180,E1 -6559.855,E2 -6559.855} C_VEL
LIN {X 0,Y 488.451,Z 532.074,A -85,B 0,C 180,E1 -6561.102,E2 -6561.102} C_VEL
LIN {X 0,Y 488.219,Z 539.328,A -85,B 0,C 180,E1 -6562.348,E2 -6562.348} C_VEL
LIN {X 0,Y 488.078,Z 544.698,A -85,B 0,C 180,E1 -6563.493,E2 -6563.493} C_VEL
LIN {X 0,Y 488.025,Z 548.985,A -85,B 0,C 180,E1 -6564.629,E2 -6564.629} C_VEL
LIN {X 0,Y 487.936,Z 552.623,A -85,B 0,C 180,E1 -6565.87,E2 -6565.87} C_VEL
LIN {X 0,Y 487.965,Z 554.504,A -85,B 0,C 180,E1 -6566.698,E2 -6566.698} C_VEL
LIN {X 0,Y 487.891,Z 556.916,A -85,B 0,C 180,E1 -6568.349,E2 -6568.349} C_VEL
LIN {X 0,Y 487.819,Z 557.754,A -85,B 0,C 180,E1 -6570,E2 -6570} C_VEL
LIN {X 0,Y 487.891,Z 556.936,A -85,B 0,C 180,E1 -6571.651,E2 -6571.651} C_VEL
LIN {X 0,Y 487.909,Z 555.941,A -85,B 0,C 180,E1 -6572.477,E2 -6572.477} C_VEL
LIN {X 0,Y 487.966,Z 554.544,A -85,B 0,C 180,E1 -6573.303,E2 -6573.303} C_VEL
LIN {X 0,Y 487.927,Z 551.597,A -85,B 0,C 180,E1 -6574.544,E2 -6574.544} C_VEL
LIN {X 0,Y 488.043,Z 547.611,A -85,B 0,C 180,E1 -6575.786,E2 -6575.786} C_VEL
LIN {X 0,Y 488.184,Z 541.472,A -85,B 0,C 180,E1 -6577.237,E2 -6577.237} C_VEL
LIN {X 0,Y 488.375,Z 534.768,A -85,B 0,C 180,E1 -6578.483,E2 -6578.483} C_VEL
LIN {X 0,Y 488.687,Z 526.453,A -85,B 0,C 180,E1 -6579.729,E2 -6579.729} C_VEL
LIN {X 0,Y 489.002,Z 517.921,A -85,B 0,C 180,E1 -6580.769,E2 -6580.769} C_VEL
LIN {X 0,Y 489.468,Z 507.39,A -85,B 0,C 180,E1 -6581.807,E2 -6581.807} C_VEL
LIN {X 0,Y 489.785,Z 495.974,A -85,B 0,C 180,E1 -6582.714,E2 -6582.714} C_VEL
LIN {X 0,Y 490.228,Z 483.607,A -85,B 0,C 180,E1 -6583.472,E2 -6583.472} C_VEL
LIN {X 0,Y 490.64,Z 471.234,A -85,B 0,C 180,E1 -6584.041,E2 -6584.041} C_VEL
LIN {X 0,Y 490.587,Z 466.239,A -85,B 0,C 180,E1 -6584.228,E2 -6584.228} C_VEL
LIN {X 0,Y 488.483,Z 452.836,A -85,B 0,C 180,E1 -6584.663,E2 -6584.663} C_VEL
LIN {X 0,Y 488.168,Z 450.611,A -85,B 0,C 180,E1 -6584.726,E2 -6584.726} C_VEL
LIN {X 0,Y 488.294,Z 442.677,A -85,B 0,C 180,E1 -6587.593,E2 -6587.593} C_VEL
LIN {X 0,Y 488.515,Z 434.095,A -85,B 0,C 180,E1 -6590.752,E2 -6590.752} C_VEL
LIN {X 0,Y 488.697,Z 426.149,A -85,B 0,C 180,E1 -6593.745,E2 -6593.745} C_VEL
LIN {X 0,Y 488.883,Z 419.084,A -85,B 0,C 180,E1 -6596.465,E2 -6596.465} C_VEL
LIN {X 0,Y 489.189,Z 410.907,A -85,B 0,C 180,E1 -6599.713,E2 -6599.713} C_VEL
LIN {X 0,Y 489.508,Z 403.922,A -85,B 0,C 180,E1 -6602.575,E2 -6602.575} C_VEL
LIN {X 0,Y 489.767,Z 397.924,A -85,B 0,C 180,E1 -6605.121,E2 -6605.121} C_VEL
LIN {X 0,Y 489.418,Z 393.522,A -85,B 0,C 180,E1 -6607.093,E2 -6607.093} C_VEL
LIN {X 0,Y 488.732,Z 389.61,A -85,B 0,C 180,E1 -6608.985,E2 -6608.985} C_VEL
LIN {X 0,Y 488.709,Z 389.611,A -85,B 0,C 180,E1 -6611.6,E2 -6611.6} C_VEL
LIN {X 0,Y 488.703,Z 389.613,A -85,B 0,C 180,E1 -6614.803,E2 -6614.803} C_VEL
LIN {X 0,Y 488.693,Z 389.613,A -85,B 0,C 180,E1 -6617.474,E2 -6617.474} C_VEL
LIN {X 0,Y 488.734,Z 389.607,A -85,B 0,C 180,E1 -6619.676,E2 -6619.676} C_VEL
LIN {X 0,Y 488.683,Z 389.614,A -85,B 0,C 180,E1 -6622.841,E2 -6622.841} C_VEL
LIN {X 0,Y 488.727,Z 389.607,A -85,B 0,C 180,E1 -6625.887,E2 -6625.887} C_VEL
LIN {X 0,Y 488.693,Z 389.613,A -85,B 0,C 180,E1 -6628.82,E2 -6628.82} C_VEL
LIN {X 0,Y 488.745,Z 389.606,A -85,B 0,C 180,E1 -6631.671,E2 -6631.671} C_VEL
LIN {X 0,Y 488.748,Z 389.605,A -85,B 0,C 180,E1 -6634.444,E2 -6634.444} C_VEL
LIN {X 0,Y 488.723,Z 389.61,A -85,B 0,C 180,E1 -6637.153,E2 -6637.153} C_VEL
LIN {X 0,Y 488.725,Z 389.609,A -85,B 0,C 180,E1 -6639.81,E2 -6639.81} C_VEL
LIN {X 0,Y 488.73,Z 389.609,A -85,B 0,C 180,E1 -6642.423,E2 -6642.423} C_VEL
LIN {X 0,Y 488.762,Z 389.604,A -85,B 0,C 180,E1 -6645,E2 -6645} C_VEL
LIN {X 0,Y 488.806,Z 389.6,A -85,B 0,C 180,E1 -6648.387,E2 -6648.387} C_VEL
LIN {X 0,Y 488.818,Z 389.597,A -85,B 0,C 180,E1 -6651.734,E2 -6651.734} C_VEL
LIN {X 0,Y 488.855,Z 389.593,A -85,B 0,C 180,E1 -6654.224,E2 -6654.224} C_VEL
LIN {X 0,Y 488.96,Z 389.58,A -85,B 0,C 180,E1 -6657.529,E2 -6657.529} C_VEL
LIN {X 0,Y 488.954,Z 389.58,A -85,B 0,C 180,E1 -6660.824,E2 -6660.824} C_VEL
LIN {X 0,Y 488.96,Z 389.58,A -85,B 0,C 180,E1 -6662.471,E2 -6662.471} C_VEL
LIN {X 0,Y 488.855,Z 389.593,A -85,B 0,C 180,E1 -6665.776,E2 -6665.776} C_VEL
LIN {X 0,Y 488.818,Z 389.597,A -85,B 0,C 180,E1 -6668.266,E2 -6668.266} C_VEL
LIN {X 0,Y 488.806,Z 389.599,A -85,B 0,C 180,E1 -6671.612,E2 -6671.612} C_VEL
LIN {X 0,Y 488.762,Z 389.604,A -85,B 0,C 180,E1 -6675,E2 -6675} C_VEL
LIN {X 0,Y 488.755,Z 389.605,A -85,B 0,C 180,E1 -6678.442,E2 -6678.442} C_VEL
LIN {X 0,Y 488.707,Z 389.611,A -85,B 0,C 180,E1 -6681.071,E2 -6681.071} C_VEL
LIN {X 0,Y 488.689,Z 389.613,A -85,B 0,C 180,E1 -6683.746,E2 -6683.746} C_VEL
LIN {X 0,Y 488.792,Z 389.601,A -85,B 0,C 180,E1 -6686.944,E2 -6686.944} C_VEL
LIN {X 0,Y 488.71,Z 389.611,A -85,B 0,C 180,E1 -6690.363,E2 -6690.363} C_VEL
LIN {X 0,Y 488.736,Z 389.607,A -85,B 0,C 180,E1 -6693.484,E2 -6693.484} C_VEL
LIN {X 0,Y 488.689,Z 389.613,A -85,B 0,C 180,E1 -6696.356,E2 -6696.356} C_VEL
LIN {X 0,Y 488.701,Z 389.613,A -85,B 0,C 180,E1 -6699.254,E2 -6699.254} C_VEL
LIN {X 0,Y 488.708,Z 389.611,A -85,B 0,C 180,E1 -6701.6,E2 -6701.6} C_VEL
LIN {X 0,Y 488.702,Z 389.612,A -85,B 0,C 180,E1 -6704.803,E2 -6704.803} C_VEL
LIN {X 0,Y 488.693,Z 389.613,A -85,B 0,C 180,E1 -6707.475,E2 -6707.475} C_VEL
LIN {X 0,Y 488.734,Z 389.606,A -85,B 0,C 180,E1 -6709.677,E2 -6709.677} C_VEL
LIN {X 0,Y 488.683,Z 389.614,A -85,B 0,C 180,E1 -6712.841,E2 -6712.841} C_VEL
LIN {X 0,Y 488.735,Z 389.606,A -85,B 0,C 180,E1 -6715.887,E2 -6715.887} C_VEL
LIN {X 0,Y 488.694,Z 389.613,A -85,B 0,C 180,E1 -6718.82,E2 -6718.82} C_VEL
LIN {X 0,Y 488.746,Z 389.604,A -85,B 0,C 180,E1 -6721.671,E2 -6721.671} C_VEL
LIN {X 0,Y 488.744,Z 389.608,A -85,B 0,C 180,E1 -6724.341,E2 -6724.341} C_VEL
LIN {X 0,Y 488.099,Z 389.692,A -85,B 0,C 180,E1 -6725.028,E2 -6725.028} C_VEL
LIN {X 0,Y 485.231,Z 390.049,A -85,B 0,C 180,E1 -6726.145,E2 -6726.145} C_VEL
LIN {X 0,Y 482.785,Z 390.349,A -85,B 0,C 180,E1 -6727.044,E2 -6727.044} C_VEL
LIN {X 0,Y 481.727,Z 390.479,A -85,B 0,C 180,E1 -6727.74,E2 -6727.74} C_VEL
LIN {X 0,Y 481.638,Z 390.489,A -85,B 0,C 180,E1 -6727.975,E2 -6727.975} C_VEL
LIN {X 0,Y 481.708,Z 390.485,A -85,B 0,C 180,E1 -6730.393,E2 -6730.393} C_VEL
LIN {X 0,Y 481.689,Z 390.484,A -85,B 0,C 180,E1 -6733.034,E2 -6733.034} C_VEL
LIN {X 0,Y 481.692,Z 390.484,A -85,B 0,C 180,E1 -6735.639,E2 -6735.639} C_VEL
LIN {X 0,Y 481.753,Z 390.477,A -85,B 0,C 180,E1 -6738.215,E2 -6738.215} C_VEL
LIN {X 0,Y 481.764,Z 390.475,A -85,B 0,C 180,E1 -6741.611,E2 -6741.611} C_VEL
LIN {X 0,Y 481.819,Z 390.469,A -85,B 0,C 180,E1 -6744.139,E2 -6744.139} C_VEL
LIN {X 0,Y 481.93,Z 390.455,A -85,B 0,C 180,E1 -6747.492,E2 -6747.492} C_VEL
LIN {X 0,Y 481.888,Z 390.46,A -85,B 0,C 180,E1 -6750.835,E2 -6750.835} C_VEL
LIN {X 0,Y 481.93,Z 390.455,A -85,B 0,C 180,E1 -6752.507,E2 -6752.507} C_VEL
LIN {X 0,Y 481.798,Z 390.472,A -85,B 0,C 180,E1 -6755.86,E2 -6755.86} C_VEL
LIN {X 0,Y 481.589,Z 390.5,A -85,B 0,C 180,E1 -6758.391,E2 -6758.391} C_VEL
LIN {X 0,Y 481.473,Z 390.854,A -85,B 0,C 180,E1 -6759.239,E2 -6759.239} C_VEL
LIN {X 0,Y 481.398,Z 394.492,A -85,B 0,C 180,E1 -6762.001,E2 -6762.001} C_VEL
LIN {X 0,Y 481.274,Z 399.14,A -85,B 0,C 180,E1 -6765.465,E2 -6765.465} C_VEL
LIN {X 0,Y 481.116,Z 403.631,A -85,B 0,C 180,E1 -6768.745,E2 -6768.745} C_VEL
LIN {X 0,Y 481.007,Z 407.349,A -85,B 0,C 180,E1 -6771.424,E2 -6771.424} C_VEL
LIN {X 0,Y 480.954,Z 411.179,A -85,B 0,C 180,E1 -6774.151,E2 -6774.151} C_VEL
LIN {X 0,Y 480.89,Z 415.12,A -85,B 0,C 180,E1 -6776.939,E2 -6776.939} C_VEL
LIN {X 0,Y 480.87,Z 416.861,A -85,B 0,C 180,E1 -6778.15,E2 -6778.15} C_VEL
LIN {X 0,Y 483.745,Z 430.74,A -85,B 0,C 180,E1 -6778.648,E2 -6778.648} C_VEL
LIN {X 0,Y 483.841,Z 437.834,A -85,B 0,C 180,E1 -6778.933,E2 -6778.933} C_VEL
LIN {X 0,Y 483.404,Z 449.67,A -85,B 0,C 180,E1 -6779.527,E2 -6779.527} C_VEL
LIN {X 0,Y 483.005,Z 460.735,A -85,B 0,C 180,E1 -6780.252,E2 -6780.252} C_VEL
LIN {X 0,Y 482.573,Z 471.88,A -85,B 0,C 180,E1 -6781.172,E2 -6781.172} C_VEL
LIN {X 0,Y 482.208,Z 480.757,A -85,B 0,C 180,E1 -6782.076,E2 -6782.076} C_VEL
LIN {X 0,Y 481.864,Z 489.508,A -85,B 0,C 180,E1 -6783.157,E2 -6783.157} C_VEL
LIN {X 0,Y 481.512,Z 497.9,A -85,B 0,C 180,E1 -6784.442,E2 -6784.442} C_VEL
LIN {X 0,Y 481.222,Z 504.729,A -85,B 0,C 180,E1 -6785.744,E2 -6785.744} C_VEL
LIN {X 0,Y 481.07,Z 509.178,A -85,B 0,C 180,E1 -6786.796,E2 -6786.796} C_VEL
LIN {X 0,Y 480.912,Z 514.442,A -85,B 0,C 180,E1 -6788.395,E2 -6788.395} C_VEL
LIN {X 0,Y 480.773,Z 518.052,A -85,B 0,C 180,E1 -6790.03,E2 -6790.03} C_VEL
LIN {X 0,Y 480.692,Z 519.623,A -85,B 0,C 180,E1 -6791.141,E2 -6791.141} C_VEL
LIN {X 0,Y 480.707,Z 520.479,A -85,B 0,C 180,E1 -6792.261,E2 -6792.261} C_VEL
LIN {X 0,Y 480.728,Z 520.608,A -85,B 0,C 180,E1 -6793.401,E2 -6793.401} C_VEL
LIN {X 0,Y 480.766,Z 520.012,A -85,B 0,C 180,E1 -6794.561,E2 -6794.561} C_VEL
LIN {X 0,Y 480.798,Z 518.628,A -85,B 0,C 180,E1 -6795.745,E2 -6795.745} C_VEL
LIN {X 0,Y 480.91,Z 515.365,A -85,B 0,C 180,E1 -6797.357,E2 -6797.357} C_VEL
LIN {X 0,Y 481.034,Z 510.768,A -85,B 0,C 180,E1 -6798.894,E2 -6798.894} C_VEL
LIN {X 0,Y 481.25,Z 504.626,A -85,B 0,C 180,E1 -6800.39,E2 -6800.39} C_VEL
LIN {X 0,Y 481.554,Z 496.975,A -85,B 0,C 180,E1 -6801.831,E2 -6801.831} C_VEL
LIN {X 0,Y 481.897,Z 489.052,A -85,B 0,C 180,E1 -6803.016,E2 -6803.016} C_VEL
LIN {X 0,Y 482.289,Z 479.071,A -85,B 0,C 180,E1 -6804.218,E2 -6804.218} C_VEL
LIN {X 0,Y 482.718,Z 469.488,A -85,B 0,C 180,E1 -6805.151,E2 -6805.151} C_VEL
LIN {X 0,Y 483.148,Z 458.598,A -85,B 0,C 180,E1 -6806.009,E2 -6806.009} C_VEL
LIN {X 0,Y 483.544,Z 446.544,A -85,B 0,C 180,E1 -6806.749,E2 -6806.749} C_VEL
LIN {X 0,Y 483.92,Z 434.753,A -85,B 0,C 180,E1 -6807.296,E2 -6807.296} C_VEL
LIN {X 0,Y 483.683,Z 430.118,A -85,B 0,C 180,E1 -6807.478,E2 -6807.478} C_VEL
LIN {X 0,Y 480.936,Z 417.263,A -85,B 0,C 180,E1 -6807.946,E2 -6807.946} C_VEL
LIN {X 0,Y 480.986,Z 412.651,A -85,B 0,C 180,E1 -6811.245,E2 -6811.245} C_VEL
LIN {X 0,Y 481.093,Z 408.847,A -85,B 0,C 180,E1 -6814.008,E2 -6814.008} C_VEL
LIN {X 0,Y 481.196,Z 404.858,A -85,B 0,C 180,E1 -6816.944,E2 -6816.944} C_VEL
LIN {X 0,Y 481.332,Z 401.464,A -85,B 0,C 180,E1 -6819.487,E2 -6819.487} C_VEL
LIN {X 0,Y 481.4,Z 397.967,A -85,B 0,C 180,E1 -6822.147,E2 -6822.147} C_VEL
LIN {X 0,Y 481.497,Z 394.559,A -85,B 0,C 180,E1 -6824.768,E2 -6824.768} C_VEL
LIN {X 0,Y 481.599,Z 390.6,A -85,B 0,C 180,E1 -6827.883,E2 -6827.883} C_VEL
LIN {X 0,Y 481.735,Z 390.483,A -85,B 0,C 180,E1 -6830.765,E2 -6830.765} C_VEL
LIN {X 0,Y 481.787,Z 390.475,A -85,B 0,C 180,E1 -6833.298,E2 -6833.298} C_VEL
LIN {X 0,Y 481.658,Z 390.49,A -85,B 0,C 180,E1 -6835.816,E2 -6835.816} C_VEL
LIN {X 0,Y 481.924,Z 390.458,A -85,B 0,C 180,E1 -6837.493,E2 -6837.493} C_VEL
LIN {X 0,Y 481.936,Z 390.455,A -85,B 0,C 180,E1 -6840,E2 -6840} C_VEL
LIN {X 0,Y 481.924,Z 390.455,A -85,B 0,C 180,E1 -6842.508,E2 -6842.508} C_VEL
LIN {X 0,Y 481.813,Z 390.472,A -85,B 0,C 180,E1 -6845.861,E2 -6845.861} C_VEL
LIN {X 0,Y 481.759,Z 390.477,A -85,B 0,C 180,E1 -6848.388,E2 -6848.388} C_VEL
LIN {X 0,Y 481.747,Z 390.478,A -85,B 0,C 180,E1 -6851.785,E2 -6851.785} C_VEL
LIN {X 0,Y 481.738,Z 390.481,A -85,B 0,C 180,E1 -6855.224,E2 -6855.224} C_VEL
LIN {X 0,Y 481.709,Z 390.483,A -85,B 0,C 180,E1 -6858.722,E2 -6858.722} C_VEL
LIN {X 0,Y 481.644,Z 390.492,A -85,B 0,C 180,E1 -6861.395,E2 -6861.395} C_VEL
LIN {X 0,Y 481.674,Z 390.485,A -85,B 0,C 180,E1 -6864.113,E2 -6864.113} C_VEL
LIN {X 0,Y 481.749,Z 390.478,A -85,B 0,C 180,E1 -6867.141,E2 -6867.141} C_VEL
LIN {X 0,Y 481.685,Z 390.487,A -85,B 0,C 180,E1 -6869.741,E2 -6869.741} C_VEL
LIN {X 0,Y 481.669,Z 390.489,A -85,B 0,C 180,E1 -6872.675,E2 -6872.675} C_VEL
LIN {X 0,Y 481.639,Z 390.493,A -85,B 0,C 180,E1 -6875.709,E2 -6875.709} C_VEL
LIN {X 0,Y 481.717,Z 390.485,A -85,B 0,C 180,E1 -6879.355,E2 -6879.355} C_VEL
LIN {X 0,Y 481.647,Z 390.493,A -85,B 0,C 180,E1 -6882.161,E2 -6882.161} C_VEL
LIN {X 0,Y 481.658,Z 390.49,A -85,B 0,C 180,E1 -6885.543,E2 -6885.543} C_VEL
LIN {X 0,Y 481.667,Z 390.488,A -85,B 0,C 180,E1 -6888.96,E2 -6888.96} C_VEL
LIN {X 0,Y 481.723,Z 390.553,A -85,B 0,C 180,E1 -6890.645,E2 -6890.645} C_VEL
LIN {X 0,Y 482.565,Z 395.855,A -85,B 0,C 180,E1 -6893.337,E2 -6893.337} C_VEL
LIN {X 0,Y 482.729,Z 400.295,A -85,B 0,C 180,E1 -6895.404,E2 -6895.404} C_VEL
LIN {X 0,Y 482.349,Z 406.993,A -85,B 0,C 180,E1 -6898.364,E2 -6898.364} C_VEL
LIN {X 0,Y 482.021,Z 413.848,A -85,B 0,C 180,E1 -6901.24,E2 -6901.24} C_VEL
LIN {X 0,Y 481.774,Z 420.807,A -85,B 0,C 180,E1 -6904.048,E2 -6904.048} C_VEL
LIN {X 0,Y 481.533,Z 429.088,A -85,B 0,C 180,E1 -6907.27,E2 -6907.27} C_VEL
LIN {X 0,Y 481.356,Z 436.109,A -85,B 0,C 180,E1 -6909.934,E2 -6909.934} C_VEL
LIN {X 0,Y 481.172,Z 444.425,A -85,B 0,C 180,E1 -6913.016,E2 -6913.016} C_VEL
LIN {X 0,Y 481.102,Z 450.19,A -85,B 0,C 180,E1 -6915.067,E2 -6915.067} C_VEL
LIN {X 0,Y 483.146,Z 463.769,A -85,B 0,C 180,E1 -6915.482,E2 -6915.482} C_VEL
LIN {X 0,Y 483.803,Z 469.385,A -85,B 0,C 180,E1 -6915.703,E2 -6915.703} C_VEL
LIN {X 0,Y 483.396,Z 481.072,A -85,B 0,C 180,E1 -6916.228,E2 -6916.228} C_VEL
LIN {X 0,Y 482.963,Z 492.326,A -85,B 0,C 180,E1 -6916.89,E2 -6916.89} C_VEL
LIN {X 0,Y 482.565,Z 503.327,A -85,B 0,C 180,E1 -6917.71,E2 -6917.71} C_VEL
LIN {X 0,Y 482.135,Z 513.508,A -85,B 0,C 180,E1 -6918.651,E2 -6918.651} C_VEL
LIN {X 0,Y 481.756,Z 522.758,A -85,B 0,C 180,E1 -6919.706,E2 -6919.706} C_VEL
LIN {X 0,Y 481.401,Z 531.77,A -85,B 0,C 180,E1 -6920.971,E2 -6920.971} C_VEL
LIN {X 0,Y 481.147,Z 539.03,A -85,B 0,C 180,E1 -6922.235,E2 -6922.235} C_VEL
LIN {X 0,Y 480.977,Z 544.92,A -85,B 0,C 180,E1 -6923.522,E2 -6923.522} C_VEL
LIN {X 0,Y 480.9,Z 550.024,A -85,B 0,C 180,E1 -6924.97,E2 -6924.97} C_VEL
LIN {X 0,Y 480.835,Z 552.341,A -85,B 0,C 180,E1 -6925.809,E2 -6925.809} C_VEL
LIN {X 0,Y 480.89,Z 554.226,A -85,B 0,C 180,E1 -6926.649,E2 -6926.649} C_VEL
LIN {X 0,Y 480.821,Z 556.643,A -85,B 0,C 180,E1 -6928.325,E2 -6928.325} C_VEL
LIN {X 0,Y 480.743,Z 557.483,A -85,B 0,C 180,E1 -6930,E2 -6930} C_VEL
LIN {X 0,Y 480.821,Z 556.667,A -85,B 0,C 180,E1 -6931.675,E2 -6931.675} C_VEL
LIN {X 0,Y 480.89,Z 554.274,A -85,B 0,C 180,E1 -6933.352,E2 -6933.352} C_VEL
LIN {X 0,Y 480.845,Z 551.326,A -85,B 0,C 180,E1 -6934.611,E2 -6934.611} C_VEL
LIN {X 0,Y 480.945,Z 547.337,A -85,B 0,C 180,E1 -6935.871,E2 -6935.871} C_VEL
LIN {X 0,Y 481.112,Z 541.196,A -85,B 0,C 180,E1 -6937.344,E2 -6937.344} C_VEL
LIN {X 0,Y 481.329,Z 534.489,A -85,B 0,C 180,E1 -6938.608,E2 -6938.608} C_VEL
LIN {X 0,Y 481.624,Z 526.17,A -85,B 0,C 180,E1 -6939.873,E2 -6939.873} C_VEL
LIN {X 0,Y 482,Z 517.634,A -85,B 0,C 180,E1 -6940.927,E2 -6940.927} C_VEL
LIN {X 0,Y 482.476,Z 507.167,A -85,B 0,C 180,E1 -6941.974,E2 -6941.974} C_VEL
LIN {X 0,Y 482.84,Z 495.68,A -85,B 0,C 180,E1 -6942.9,E2 -6942.9} C_VEL
LIN {X 0,Y 483.322,Z 483.307,A -85,B 0,C 180,E1 -6943.668,E2 -6943.668} C_VEL
LIN {X 0,Y 483.751,Z 470.931,A -85,B 0,C 180,E1 -6944.245,E2 -6944.245} C_VEL
LIN {X 0,Y 483.595,Z 466.685,A -85,B 0,C 180,E1 -6944.411,E2 -6944.411} C_VEL
LIN {X 0,Y 481.515,Z 453.241,A -85,B 0,C 180,E1 -6944.863,E2 -6944.863} C_VEL
LIN {X 0,Y 481.089,Z 450.355,A -85,B 0,C 180,E1 -6944.948,E2 -6944.948} C_VEL
LIN {X 0,Y 481.231,Z 442.461,A -85,B 0,C 180,E1 -6947.86,E2 -6947.86} C_VEL
LIN {X 0,Y 481.465,Z 434.361,A -85,B 0,C 180,E1 -6950.898,E2 -6950.898} C_VEL
LIN {X 0,Y 481.655,Z 425.947,A -85,B 0,C 180,E1 -6954.114,E2 -6954.114} C_VEL
LIN {X 0,Y 481.913,Z 418.185,A -85,B 0,C 180,E1 -6957.177,E2 -6957.177} C_VEL
LIN {X 0,Y 482.245,Z 410.768,A -85,B 0,C 180,E1 -6960.185,E2 -6960.185} C_VEL
LIN {X 0,Y 482.559,Z 403.8,A -85,B 0,C 180,E1 -6963.103,E2 -6963.103} C_VEL
LIN {X 0,Y 482.764,Z 398.014,A -85,B 0,C 180,E1 -6965.613,E2 -6965.613} C_VEL
LIN {X 0,Y 482.183,Z 393.403,A -85,B 0,C 180,E1 -6967.746,E2 -6967.746} C_VEL
LIN {X 0,Y 481.691,Z 390.487,A -85,B 0,C 180,E1 -6969.183,E2 -6969.183} C_VEL
LIN {X 0,Y 481.649,Z 390.492,A -85,B 0,C 180,E1 -6972.161,E2 -6972.161} C_VEL
LIN {X 0,Y 481.656,Z 390.49,A -85,B 0,C 180,E1 -6975.542,E2 -6975.542} C_VEL
LIN {X 0,Y 481.657,Z 390.489,A -85,B 0,C 180,E1 -6978.958,E2 -6978.958} C_VEL
LIN {X 0,Y 481.657,Z 390.489,A -85,B 0,C 180,E1 -6981.992,E2 -6981.992} C_VEL
LIN {X 0,Y 481.688,Z 390.487,A -85,B 0,C 180,E1 -6985.318,E2 -6985.318} C_VEL
LIN {X 0,Y 481.645,Z 390.49,A -85,B 0,C 180,E1 -6988.311,E2 -6988.311} C_VEL
LIN {X 0,Y 481.701,Z 390.485,A -85,B 0,C 180,E1 -6991.218,E2 -6991.218} C_VEL
LIN {X 0,Y 481.701,Z 390.483,A -85,B 0,C 180,E1 -6994.043,E2 -6994.043} C_VEL
LIN {X 0,Y 481.675,Z 390.487,A -85,B 0,C 180,E1 -6996.812,E2 -6996.812} C_VEL
LIN {X 0,Y 481.696,Z 390.486,A -85,B 0,C 180,E1 -6999.503,E2 -6999.503} C_VEL
LIN {X 0,Y 481.705,Z 390.483,A -85,B 0,C 180,E1 -7002.158,E2 -7002.158} C_VEL
LIN {X 0,Y 481.743,Z 390.48,A -85,B 0,C 180,E1 -7004.776,E2 -7004.776} C_VEL
LIN {X 0,Y 481.751,Z 390.477,A -85,B 0,C 180,E1 -7008.215,E2 -7008.215} C_VEL
LIN {X 0,Y 481.763,Z 390.476,A -85,B 0,C 180,E1 -7011.612,E2 -7011.612} C_VEL
LIN {X 0,Y 481.816,Z 390.469,A -85,B 0,C 180,E1 -7014.14,E2 -7014.14} C_VEL
LIN {X 0,Y 481.927,Z 390.457,A -85,B 0,C 180,E1 -7017.492,E2 -7017.492} C_VEL
LIN {X 0,Y 481.905,Z 390.459,A -85,B 0,C 180,E1 -7020.836,E2 -7020.836} C_VEL
LIN {X 0,Y 481.927,Z 390.457,A -85,B 0,C 180,E1 -7022.507,E2 -7022.507} C_VEL
LIN {X 0,Y 481.816,Z 390.469,A -85,B 0,C 180,E1 -7025.86,E2 -7025.86} C_VEL
LIN {X 0,Y 481.763,Z 390.476,A -85,B 0,C 180,E1 -7028.388,E2 -7028.388} C_VEL
LIN {X 0,Y 481.751,Z 390.477,A -85,B 0,C 180,E1 -7031.785,E2 -7031.785} C_VEL
LIN {X 0,Y 481.743,Z 390.479,A -85,B 0,C 180,E1 -7035.224,E2 -7035.224} C_VEL
LIN {X 0,Y 481.712,Z 390.483,A -85,B 0,C 180,E1 -7038.722,E2 -7038.722} C_VEL
LIN {X 0,Y 481.646,Z 390.491,A -85,B 0,C 180,E1 -7041.395,E2 -7041.395} C_VEL
LIN {X 0,Y 481.674,Z 390.488,A -85,B 0,C 180,E1 -7044.113,E2 -7044.113} C_VEL
LIN {X 0,Y 481.747,Z 390.479,A -85,B 0,C 180,E1 -7047.139,E2 -7047.139} C_VEL
LIN {X 0,Y 481.679,Z 390.486,A -85,B 0,C 180,E1 -7049.741,E2 -7049.741} C_VEL
LIN {X 0,Y 481.673,Z 390.488,A -85,B 0,C 180,E1 -7052.674,E2 -7052.674} C_VEL
LIN {X 0,Y 481.643,Z 390.491,A -85,B 0,C 180,E1 -7055.709,E2 -7055.709} C_VEL
LIN {X 0,Y 481.671,Z 390.488,A -85,B 0,C 180,E1 -7058.859,E2 -7058.859} C_VEL
LIN {X 0,Y 481.653,Z 390.49,A -85,B 0,C 180,E1 -7061.913,E2 -7061.913} C_VEL
LIN {X 0,Y 481.655,Z 390.49,A -85,B 0,C 180,E1 -7064.458,E2 -7064.458} C_VEL
LIN {X 0,Y 481.649,Z 390.49,A -85,B 0,C 180,E1 -7067.839,E2 -7067.839} C_VEL
LIN {X 0,Y 481.681,Z 390.486,A -85,B 0,C 180,E1 -7070.651,E2 -7070.651} C_VEL
LIN {X 0,Y 481.632,Z 390.492,A -85,B 0,C 180,E1 -7073.376,E2 -7073.376} C_VEL
LIN {X 0,Y 481.711,Z 390.484,A -85,B 0,C 180,E1 -7076.33,E2 -7076.33} C_VEL
LIN {X 0,Y 481.652,Z 390.489,A -85,B 0,C 180,E1 -7079.417,E2 -7079.417} C_VEL
LIN {X 0,Y 481.702,Z 390.485,A -85,B 0,C 180,E1 -7082.168,E2 -7082.168} C_VEL
LIN {X 0,Y 481.72,Z 390.481,A -85,B 0,C 180,E1 -7084.97,E2 -7084.97} C_VEL
LIN {X 0,Y 481.638,Z 390.489,A -85,B 0,C 180,E1 -7087.975,E2 -7087.975} C_VEL
LIN {X 0,Y 480.97,Z 390.576,A -85,B 0,C 180,E1 -7088.673,E2 -7088.673} C_VEL
LIN {X 0,Y 478.145,Z 390.926,A -85,B 0,C 180,E1 -7089.808,E2 -7089.808} C_VEL
LIN {X 0,Y 475.761,Z 391.224,A -85,B 0,C 180,E1 -7090.722,E2 -7090.722} C_VEL
LIN {X 0,Y 474.739,Z 391.35,A -85,B 0,C 180,E1 -7091.428,E2 -7091.428} C_VEL
LIN {X 0,Y 474.657,Z 391.361,A -85,B 0,C 180,E1 -7091.667,E2 -7091.667} C_VEL
LIN {X 0,Y 474.702,Z 391.356,A -85,B 0,C 180,E1 -7094.544,E2 -7094.544} C_VEL
LIN {X 0,Y 474.707,Z 391.355,A -85,B 0,C 180,E1 -7098.037,E2 -7098.037} C_VEL
LIN {X 0,Y 474.729,Z 391.352,A -85,B 0,C 180,E1 -7101.486,E2 -7101.486} C_VEL
LIN {X 0,Y 474.782,Z 391.346,A -85,B 0,C 180,E1 -7104.052,E2 -7104.052} C_VEL
LIN {X 0,Y 474.896,Z 391.331,A -85,B 0,C 180,E1 -7107.455,E2 -7107.455} C_VEL
LIN {X 0,Y 474.914,Z 391.329,A -85,B 0,C 180,E1 -7110,E2 -7110} C_VEL
LIN {X 0,Y 474.896,Z 391.332,A -85,B 0,C 180,E1 -7112.544,E2 -7112.544} C_VEL
LIN {X 0,Y 474.757,Z 391.349,A -85,B 0,C 180,E1 -7115.947,E2 -7115.947} C_VEL
LIN {X 0,Y 474.521,Z 391.38,A -85,B 0,C 180,E1 -7118.517,E2 -7118.517} C_VEL
LIN {X 0,Y 474.425,Z 391.85,A -85,B 0,C 180,E1 -7119.378,E2 -7119.378} C_VEL
LIN {X 0,Y 474.333,Z 395.358,A -85,B 0,C 180,E1 -7122.069,E2 -7122.069} C_VEL
LIN {X 0,Y 474.202,Z 399.99,A -85,B 0,C 180,E1 -7125.561,E2 -7125.561} C_VEL
LIN {X 0,Y 474.097,Z 403.86,A -85,B 0,C 180,E1 -7128.425,E2 -7128.425} C_VEL
LIN {X 0,Y 473.922,Z 408.459,A -85,B 0,C 180,E1 -7131.761,E2 -7131.761} C_VEL
LIN {X 0,Y 473.864,Z 412.31,A -85,B 0,C 180,E1 -7134.536,E2 -7134.536} C_VEL
LIN {X 0,Y 473.824,Z 417.105,A -85,B 0,C 180,E1 -7137.914,E2 -7137.914} C_VEL
LIN {X 0,Y 476.872,Z 431.749,A -85,B 0,C 180,E1 -7138.468,E2 -7138.468} C_VEL
LIN {X 0,Y 476.908,Z 439.551,A -85,B 0,C 180,E1 -7138.796,E2 -7138.796} C_VEL
LIN {X 0,Y 476.419,Z 451.29,A -85,B 0,C 180,E1 -7139.415,E2 -7139.415} C_VEL
LIN {X 0,Y 475.965,Z 463.496,A -85,B 0,C 180,E1 -7140.257,E2 -7140.257} C_VEL
LIN {X 0,Y 475.545,Z 473.684,A -85,B 0,C 180,E1 -7141.148,E2 -7141.148} C_VEL
LIN {X 0,Y 475.147,Z 483.189,A -85,B 0,C 180,E1 -7142.173,E2 -7142.173} C_VEL
LIN {X 0,Y 474.764,Z 492.407,A -85,B 0,C 180,E1 -7143.395,E2 -7143.395} C_VEL
LIN {X 0,Y 474.427,Z 499.294,A -85,B 0,C 180,E1 -7144.514,E2 -7144.514} C_VEL
LIN {X 0,Y 474.144,Z 505.967,A -85,B 0,C 180,E1 -7145.851,E2 -7145.851} C_VEL
LIN {X 0,Y 473.918,Z 512.053,A -85,B 0,C 180,E1 -7147.445,E2 -7147.445} C_VEL
LIN {X 0,Y 473.783,Z 516.429,A -85,B 0,C 180,E1 -7149.021,E2 -7149.021} C_VEL
LIN {X 0,Y 473.714,Z 517.719,A -85,B 0,C 180,E1 -7149.638,E2 -7149.638} C_VEL
LIN {X 0,Y 473.641,Z 519.551,A -85,B 0,C 180,E1 -7150.821,E2 -7150.821} C_VEL
LIN {X 0,Y 473.608,Z 520.665,A -85,B 0,C 180,E1 -7152.101,E2 -7152.101} C_VEL
LIN {X 0,Y 473.633,Z 520.889,A -85,B 0,C 180,E1 -7153.357,E2 -7153.357} C_VEL
LIN {X 0,Y 473.672,Z 520.283,A -85,B 0,C 180,E1 -7154.587,E2 -7154.587} C_VEL
LIN {X 0,Y 473.707,Z 518.897,A -85,B 0,C 180,E1 -7155.789,E2 -7155.789} C_VEL
LIN {X 0,Y 473.83,Z 515.567,A -85,B 0,C 180,E1 -7157.452,E2 -7157.452} C_VEL
LIN {X 0,Y 473.945,Z 512.084,A -85,B 0,C 180,E1 -7158.667,E2 -7158.667} C_VEL
LIN {X 0,Y 474.128,Z 506.577,A -85,B 0,C 180,E1 -7160.126,E2 -7160.126} C_VEL
LIN {X 0,Y 474.42,Z 499.757,A -85,B 0,C 180,E1 -7161.524,E2 -7161.524} C_VEL
LIN {X 0,Y 474.788,Z 491.373,A -85,B 0,C 180,E1 -7162.875,E2 -7162.875} C_VEL
LIN {X 0,Y 475.224,Z 481.894,A -85,B 0,C 180,E1 -7164.101,E2 -7164.101} C_VEL
LIN {X 0,Y 475.736,Z 471.223,A -85,B 0,C 180,E1 -7165.196,E2 -7165.196} C_VEL
LIN {X 0,Y 476.214,Z 459.677,A -85,B 0,C 180,E1 -7166.143,E2 -7166.143} C_VEL
LIN {X 0,Y 476.629,Z 448.245,A -85,B 0,C 180,E1 -7166.873,E2 -7166.873} C_VEL
LIN {X 0,Y 477.084,Z 434.804,A -85,B 0,C 180,E1 -7167.515,E2 -7167.515} C_VEL
LIN {X 0,Y 476.552,Z 429.527,A -85,B 0,C 180,E1 -7167.732,E2 -7167.732} C_VEL
LIN {X 0,Y 473.855,Z 417.566,A -85,B 0,C 180,E1 -7168.167,E2 -7168.167} C_VEL
LIN {X 0,Y 473.912,Z 413.603,A -85,B 0,C 180,E1 -7171.038,E2 -7171.038} C_VEL
LIN {X 0,Y 474.001,Z 410.122,A -85,B 0,C 180,E1 -7173.589,E2 -7173.589} C_VEL
LIN {X 0,Y 474.149,Z 405.845,A -85,B 0,C 180,E1 -7176.776,E2 -7176.776} C_VEL
LIN {X 0,Y 474.271,Z 401.48,A -85,B 0,C 180,E1 -7180.073,E2 -7180.073} C_VEL
LIN {X 0,Y 474.359,Z 398.007,A -85,B 0,C 180,E1 -7182.764,E2 -7182.764} C_VEL
LIN {X 0,Y 474.437,Z 394.617,A -85,B 0,C 180,E1 -7185.414,E2 -7185.414} C_VEL
LIN {X 0,Y 474.563,Z 391.376,A -85,B 0,C 180,E1 -7188.034,E2 -7188.034} C_VEL
LIN {X 0,Y 474.7,Z 391.36,A -85,B 0,C 180,E1 -7190.627,E2 -7190.627} C_VEL
LIN {X 0,Y 474.747,Z 391.352,A -85,B 0,C 180,E1 -7193.199,E2 -7193.199} C_VEL
LIN {X 0,Y 474.618,Z 391.367,A -85,B 0,C 180,E1 -7195.754,E2 -7195.754} C_VEL
LIN {X 0,Y 474.891,Z 391.334,A -85,B 0,C 180,E1 -7197.455,E2 -7197.455} C_VEL
LIN {X 0,Y 474.873,Z 391.336,A -85,B 0,C 180,E1 -7200.848,E2 -7200.848} C_VEL
LIN {X 0,Y 474.89,Z 391.332,A -85,B 0,C 180,E1 -7202.545,E2 -7202.545} C_VEL
LIN {X 0,Y 474.775,Z 391.348,A -85,B 0,C 180,E1 -7205.948,E2 -7205.948} C_VEL
LIN {X 0,Y 474.724,Z 391.353,A -85,B 0,C 180,E1 -7208.514,E2 -7208.514} C_VEL
LIN {X 0,Y 474.7,Z 391.357,A -85,B 0,C 180,E1 -7211.963,E2 -7211.963} C_VEL
LIN {X 0,Y 474.696,Z 391.357,A -85,B 0,C 180,E1 -7215.456,E2 -7215.456} C_VEL
LIN {X 0,Y 474.662,Z 391.361,A -85,B 0,C 180,E1 -7219.01,E2 -7219.01} C_VEL
LIN {X 0,Y 474.587,Z 391.371,A -85,B 0,C 180,E1 -7221.729,E2 -7221.729} C_VEL
LIN {X 0,Y 474.656,Z 391.36,A -85,B 0,C 180,E1 -7224.493,E2 -7224.493} C_VEL
LIN {X 0,Y 474.695,Z 391.356,A -85,B 0,C 180,E1 -7227.339,E2 -7227.339} C_VEL
LIN {X 0,Y 474.606,Z 391.369,A -85,B 0,C 180,E1 -7230.812,E2 -7230.812} C_VEL
LIN {X 0,Y 474.635,Z 391.367,A -85,B 0,C 180,E1 -7233.985,E2 -7233.985} C_VEL
LIN {X 0,Y 474.573,Z 391.374,A -85,B 0,C 180,E1 -7236.901,E2 -7236.901} C_VEL
LIN {X 0,Y 474.653,Z 391.364,A -85,B 0,C 180,E1 -7239.652,E2 -7239.652} C_VEL
LIN {X 0,Y 474.613,Z 391.368,A -85,B 0,C 180,E1 -7242.935,E2 -7242.935} C_VEL
LIN {X 0,Y 474.607,Z 391.368,A -85,B 0,C 180,E1 -7245.896,E2 -7245.896} C_VEL
LIN {X 0,Y 474.64,Z 391.364,A -85,B 0,C 180,E1 -7249.039,E2 -7249.039} C_VEL
LIN {X 0,Y 474.655,Z 391.376,A -85,B 0,C 180,E1 -7250.349,E2 -7250.349} C_VEL
LIN {X 0,Y 475.464,Z 396.413,A -85,B 0,C 180,E1 -7252.958,E2 -7252.958} C_VEL
LIN {X 0,Y 475.758,Z 400.204,A -85,B 0,C 180,E1 -7254.823,E2 -7254.823} C_VEL
LIN {X 0,Y 475.397,Z 406.905,A -85,B 0,C 180,E1 -7257.846,E2 -7257.846} C_VEL
LIN {X 0,Y 475.064,Z 413.747,A -85,B 0,C 180,E1 -7260.79,E2 -7260.79} C_VEL
LIN {X 0,Y 474.712,Z 421.797,A -85,B 0,C 180,E1 -7264.104,E2 -7264.104} C_VEL
LIN {X 0,Y 474.471,Z 429.984,A -85,B 0,C 180,E1 -7267.349,E2 -7267.349} C_VEL
LIN {X 0,Y 474.266,Z 437.063,A -85,B 0,C 180,E1 -7270.073,E2 -7270.073} C_VEL
LIN {X 0,Y 474.101,Z 445.346,A -85,B 0,C 180,E1 -7273.198,E2 -7273.198} C_VEL
LIN {X 0,Y 474.052,Z 449.95,A -85,B 0,C 180,E1 -7274.84,E2 -7274.84} C_VEL
LIN {X 0,Y 476.066,Z 463.482,A -85,B 0,C 180,E1 -7275.261,E2 -7275.261} C_VEL
LIN {X 0,Y 476.869,Z 470.391,A -85,B 0,C 180,E1 -7275.545,E2 -7275.545} C_VEL
LIN {X 0,Y 476.42,Z 482.758,A -85,B 0,C 180,E1 -7276.131,E2 -7276.131} C_VEL
LIN {X 0,Y 475.912,Z 494.704,A -85,B 0,C 180,E1 -7276.877,E2 -7276.877} C_VEL
LIN {X 0,Y 475.448,Z 505.819,A -85,B 0,C 180,E1 -7277.771,E2 -7277.771} C_VEL
LIN {X 0,Y 475.083,Z 515.183,A -85,B 0,C 180,E1 -7278.697,E2 -7278.697} C_VEL
LIN {X 0,Y 474.624,Z 524.1,A -85,B 0,C 180,E1 -7279.765,E2 -7279.765} C_VEL
LIN {X 0,Y 474.288,Z 532.813,A -85,B 0,C 180,E1 -7281.049,E2 -7281.049} C_VEL
LIN {X 0,Y 474.038,Z 539.774,A -85,B 0,C 180,E1 -7282.332,E2 -7282.332} C_VEL
LIN {X 0,Y 473.88,Z 545.101,A -85,B 0,C 180,E1 -7283.547,E2 -7283.547} C_VEL
LIN {X 0,Y 473.831,Z 549.741,A -85,B 0,C 180,E1 -7284.895,E2 -7284.895} C_VEL
LIN {X 0,Y 473.741,Z 552.06,A -85,B 0,C 180,E1 -7285.747,E2 -7285.747} C_VEL
LIN {X 0,Y 473.797,Z 553.947,A -85,B 0,C 180,E1 -7286.599,E2 -7286.599} C_VEL
LIN {X 0,Y 473.742,Z 555.359,A -85,B 0,C 180,E1 -7287.45,E2 -7287.45} C_VEL
LIN {X 0,Y 473.724,Z 556.37,A -85,B 0,C 180,E1 -7288.3,E2 -7288.3} C_VEL
LIN {X 0,Y 473.688,Z 556.988,A -85,B 0,C 180,E1 -7289.15,E2 -7289.15} C_VEL
LIN {X 0,Y 473.669,Z 557.212,A -85,B 0,C 180,E1 -7290,E2 -7290} C_VEL
LIN {X 0,Y 473.688,Z 557.001,A -85,B 0,C 180,E1 -7290.85,E2 -7290.85} C_VEL
LIN {X 0,Y 473.724,Z 556.397,A -85,B 0,C 180,E1 -7291.701,E2 -7291.701} C_VEL
LIN {X 0,Y 473.742,Z 555.402,A -85,B 0,C 180,E1 -7292.551,E2 -7292.551} C_VEL
LIN {X 0,Y 473.797,Z 554.003,A -85,B 0,C 180,E1 -7293.402,E2 -7293.402} C_VEL
LIN {X 0,Y 473.767,Z 551.055,A -85,B 0,C 180,E1 -7294.68,E2 -7294.68} C_VEL
LIN {X 0,Y 473.851,Z 547.063,A -85,B 0,C 180,E1 -7295.96,E2 -7295.96} C_VEL
LIN {X 0,Y 474.024,Z 540.919,A -85,B 0,C 180,E1 -7297.454,E2 -7297.454} C_VEL
LIN {X 0,Y 474.281,Z 534.21,A -85,B 0,C 180,E1 -7298.737,E2 -7298.737} C_VEL
LIN {X 0,Y 474.58,Z 525.885,A -85,B 0,C 180,E1 -7300.021,E2 -7300.021} C_VEL
LIN {X 0,Y 474.995,Z 517.34,A -85,B 0,C 180,E1 -7301.09,E2 -7301.09} C_VEL
LIN {X 0,Y 475.492,Z 507.082,A -85,B 0,C 180,E1 -7302.133,E2 -7302.133} C_VEL
LIN {X 0,Y 475.825,Z 496.649,A -85,B 0,C 180,E1 -7302.996,E2 -7302.996} C_VEL
LIN {X 0,Y 476.318,Z 484.93,A -85,B 0,C 180,E1 -7303.764,E2 -7303.764} C_VEL
LIN {X 0,Y 476.771,Z 473.158,A -85,B 0,C 180,E1 -7304.349,E2 -7304.349} C_VEL
LIN {X 0,Y 476.907,Z 469.286,A -85,B 0,C 180,E1 -7304.509,E2 -7304.509} C_VEL
LIN {X 0,Y 474.98,Z 456.038,A -85,B 0,C 180,E1 -7304.993,E2 -7304.993} C_VEL
LIN {X 0,Y 474.031,Z 450.127,A -85,B 0,C 180,E1 -7305.175,E2 -7305.175} C_VEL
LIN {X 0,Y 474.228,Z 441.341,A -85,B 0,C 180,E1 -7308.473,E2 -7308.473} C_VEL
LIN {X 0,Y 474.438,Z 432.822,A -85,B 0,C 180,E1 -7311.736,E2 -7311.736} C_VEL
LIN {X 0,Y 474.704,Z 424.615,A -85,B 0,C 180,E1 -7314.957,E2 -7314.957} C_VEL
LIN {X 0,Y 474.986,Z 416.421,A -85,B 0,C 180,E1 -7318.26,E2 -7318.26} C_VEL
LIN {X 0,Y 475.301,Z 409.465,A -85,B 0,C 180,E1 -7321.166,E2 -7321.166} C_VEL
LIN {X 0,Y 475.676,Z 402.487,A -85,B 0,C 180,E1 -7324.168,E2 -7324.168} C_VEL
LIN {X 0,Y 475.684,Z 397.901,A -85,B 0,C 180,E1 -7326.227,E2 -7326.227} C_VEL
LIN {X 0,Y 474.784,Z 392.147,A -85,B 0,C 180,E1 -7328.984,E2 -7328.984} C_VEL
LIN {X 0,Y 474.67,Z 391.361,A -85,B 0,C 180,E1 -7329.406,E2 -7329.406} C_VEL
LIN {X 0,Y 474.626,Z 391.367,A -85,B 0,C 180,E1 -7332.237,E2 -7332.237} C_VEL
LIN {X 0,Y 474.618,Z 391.366,A -85,B 0,C 180,E1 -7335.298,E2 -7335.298} C_VEL
LIN {X 0,Y 474.621,Z 391.365,A -85,B 0,C 180,E1 -7338.214,E2 -7338.214} C_VEL
LIN {X 0,Y 474.613,Z 391.368,A -85,B 0,C 180,E1 -7341.543,E2 -7341.543} C_VEL
LIN {X 0,Y 474.627,Z 391.365,A -85,B 0,C 180,E1 -7344.726,E2 -7344.726} C_VEL
LIN {X 0,Y 474.635,Z 391.364,A -85,B 0,C 180,E1 -7347.788,E2 -7347.788} C_VEL
LIN {X 0,Y 474.625,Z 391.365,A -85,B 0,C 180,E1 -7350.884,E2 -7350.884} C_VEL
LIN {X 0,Y 474.661,Z 391.362,A -85,B 0,C 180,E1 -7353.628,E2 -7353.628} C_VEL
LIN {X 0,Y 474.636,Z 391.364,A -85,B 0,C 180,E1 -7356.641,E2 -7356.641} C_VEL
LIN {X 0,Y 474.655,Z 391.36,A -85,B 0,C 180,E1 -7360.089,E2 -7360.089} C_VEL
LIN {X 0,Y 474.648,Z 391.362,A -85,B 0,C 180,E1 -7362.774,E2 -7362.774} C_VEL
LIN {X 0,Y 474.648,Z 391.363,A -85,B 0,C 180,E1 -7365.421,E2 -7365.421} C_VEL
LIN {X 0,Y 474.704,Z 391.355,A -85,B 0,C 180,E1 -7368.037,E2 -7368.037} C_VEL
LIN {X 0,Y 474.729,Z 391.354,A -85,B 0,C 180,E1 -7371.486,E2 -7371.486} C_VEL
LIN {X 0,Y 474.779,Z 391.345,A -85,B 0,C 180,E1 -7374.052,E2 -7374.052} C_VEL
LIN {X 0,Y 474.893,Z 391.333,A -85,B 0,C 180,E1 -7377.455,E2 -7377.455} C_VEL
LIN {X 0,Y 474.912,Z 391.329,A -85,B 0,C 180,E1 -7380,E2 -7380} C_VEL
LIN {X 0,Y 474.893,Z 391.333,A -85,B 0,C 180,E1 -7382.545,E2 -7382.545} C_VEL
LIN {X 0,Y 474.779,Z 391.345,A -85,B 0,C 180,E1 -7385.948,E2 -7385.948} C_VEL
LIN {X 0,Y 474.729,Z 391.354,A -85,B 0,C 180,E1 -7388.513,E2 -7388.513} C_VEL
LIN {X 0,Y 474.704,Z 391.355,A -85,B 0,C 180,E1 -7391.962,E2 -7391.962} C_VEL
LIN {X 0,Y 474.7,Z 391.356,A -85,B 0,C 180,E1 -7395.456,E2 -7395.456} C_VEL
LIN {X 0,Y 474.665,Z 391.362,A -85,B 0,C 180,E1 -7399.01,E2 -7399.01} C_VEL
LIN {X 0,Y 474.589,Z 391.369,A -85,B 0,C 180,E1 -7401.729,E2 -7401.729} C_VEL
LIN {X 0,Y 474.657,Z 391.361,A -85,B 0,C 180,E1 -7404.493,E2 -7404.493} C_VEL
LIN {X 0,Y 474.681,Z 391.359,A -85,B 0,C 180,E1 -7407.334,E2 -7407.334} C_VEL
LIN {X 0,Y 474.605,Z 391.369,A -85,B 0,C 180,E1 -7410.81,E2 -7410.81} C_VEL
LIN {X 0,Y 474.639,Z 391.362,A -85,B 0,C 180,E1 -7413.984,E2 -7413.984} C_VEL
LIN {X 0,Y 474.576,Z 391.373,A -85,B 0,C 180,E1 -7416.9,E2 -7416.9} C_VEL
LIN {X 0,Y 474.618,Z 391.365,A -85,B 0,C 180,E1 -7419.646,E2 -7419.646} C_VEL
LIN {X 0,Y 474.615,Z 391.368,A -85,B 0,C 180,E1 -7422.934,E2 -7422.934} C_VEL
LIN {X 0,Y 474.607,Z 391.367,A -85,B 0,C 180,E1 -7425.895,E2 -7425.895} C_VEL
LIN {X 0,Y 474.629,Z 391.365,A -85,B 0,C 180,E1 -7429.041,E2 -7429.041} C_VEL
LIN {X 0,Y 474.611,Z 391.366,A -85,B 0,C 180,E1 -7431.704,E2 -7431.704} C_VEL
LIN {X 0,Y 474.63,Z 391.366,A -85,B 0,C 180,E1 -7434.726,E2 -7434.726} C_VEL
LIN {X 0,Y 474.637,Z 391.363,A -85,B 0,C 180,E1 -7437.788,E2 -7437.788} C_VEL
LIN {X 0,Y 474.626,Z 391.366,A -85,B 0,C 180,E1 -7440.885,E2 -7440.885} C_VEL
LIN {X 0,Y 474.662,Z 391.36,A -85,B 0,C 180,E1 -7443.628,E2 -7443.628} C_VEL
LIN {X 0,Y 474.638,Z 391.365,A -85,B 0,C 180,E1 -7446.641,E2 -7446.641} C_VEL
LIN {X 0,Y 474.657,Z 391.361,A -85,B 0,C 180,E1 -7450.089,E2 -7450.089} C_VEL
LIN {X 0,Y 474.657,Z 391.361,A -85,B 0,C 180,E1 -7451.667,E2 -7451.667} C_VEL
LIN {X 0,Y 473.992,Z 391.446,A -85,B 0,C 180,E1 -7452.376,E2 -7452.376} C_VEL
LIN {X 0,Y 471.142,Z 391.802,A -85,B 0,C 180,E1 -7453.527,E2 -7453.527} C_VEL
LIN {X 0,Y 468.727,Z 392.101,A -85,B 0,C 180,E1 -7454.456,E2 -7454.456} C_VEL
LIN {X 0,Y 467.686,Z 392.229,A -85,B 0,C 180,E1 -7455.173,E2 -7455.173} C_VEL
LIN {X 0,Y 467.599,Z 392.239,A -85,B 0,C 180,E1 -7455.416,E2 -7455.416} C_VEL
LIN {X 0,Y 467.654,Z 392.234,A -85,B 0,C 180,E1 -7458.734,E2 -7458.734} C_VEL
LIN {X 0,Y 467.751,Z 392.223,A -85,B 0,C 180,E1 -7462.228,E2 -7462.228} C_VEL
LIN {X 0,Y 467.726,Z 392.224,A -85,B 0,C 180,E1 -7464.827,E2 -7464.827} C_VEL
LIN {X 0,Y 467.861,Z 392.207,A -85,B 0,C 180,E1 -7467.417,E2 -7467.417} C_VEL
LIN {X 0,Y 467.885,Z 392.205,A -85,B 0,C 180,E1 -7470,E2 -7470} C_VEL
LIN {X 0,Y 467.862,Z 392.208,A -85,B 0,C 180,E1 -7472.583,E2 -7472.583} C_VEL
LIN {X 0,Y 467.718,Z 392.226,A -85,B 0,C 180,E1 -7476.037,E2 -7476.037} C_VEL
LIN {X 0,Y 467.445,Z 392.262,A -85,B 0,C 180,E1 -7478.647,E2 -7478.647} C_VEL
LIN {X 0,Y 467.365,Z 392.856,A -85,B 0,C 180,E1 -7479.521,E2 -7479.521} C_VEL
LIN {X 0,Y 467.26,Z 396.244,A -85,B 0,C 180,E1 -7482.155,E2 -7482.155} C_VEL
LIN {X 0,Y 467.121,Z 400.856,A -85,B 0,C 180,E1 -7485.655,E2 -7485.655} C_VEL
LIN {X 0,Y 467.01,Z 404.726,A -85,B 0,C 180,E1 -7488.543,E2 -7488.543} C_VEL
LIN {X 0,Y 466.844,Z 409.582,A -85,B 0,C 180,E1 -7492.108,E2 -7492.108} C_VEL
LIN {X 0,Y 466.791,Z 414.127,A -85,B 0,C 180,E1 -7495.397,E2 -7495.397} C_VEL
LIN {X 0,Y 466.735,Z 417.357,A -85,B 0,C 180,E1 -7497.7,E2 -7497.7} C_VEL
LIN {X 0,Y 469.602,Z 430.532,A -85,B 0,C 180,E1 -7498.187,E2 -7498.187} C_VEL
LIN {X 0,Y 470.165,Z 435.319,A -85,B 0,C 180,E1 -7498.393,E2 -7498.393} C_VEL
LIN {X 0,Y 469.668,Z 448.543,A -85,B 0,C 180,E1 -7499.037,E2 -7499.037} C_VEL
LIN {X 0,Y 469.17,Z 460.548,A -85,B 0,C 180,E1 -7499.825,E2 -7499.825} C_VEL
LIN {X 0,Y 468.722,Z 471.551,A -85,B 0,C 180,E1 -7500.748,E2 -7500.748} C_VEL
LIN {X 0,Y 468.237,Z 481.814,A -85,B 0,C 180,E1 -7501.816,E2 -7501.816} C_VEL
LIN {X 0,Y 467.81,Z 490.902,A -85,B 0,C 180,E1 -7502.995,E2 -7502.995} C_VEL
LIN {X 0,Y 467.445,Z 498.567,A -85,B 0,C 180,E1 -7504.216,E2 -7504.216} C_VEL
LIN {X 0,Y 467.097,Z 505.85,A -85,B 0,C 180,E1 -7505.66,E2 -7505.66} C_VEL
LIN {X 0,Y 466.896,Z 511.384,A -85,B 0,C 180,E1 -7507.081,E2 -7507.081} C_VEL
LIN {X 0,Y 466.746,Z 515.484,A -85,B 0,C 180,E1 -7508.465,E2 -7508.465} C_VEL
LIN {X 0,Y 466.614,Z 518.367,A -85,B 0,C 180,E1 -7509.812,E2 -7509.812} C_VEL
LIN {X 0,Y 466.527,Z 520.561,A -85,B 0,C 180,E1 -7511.516,E2 -7511.516} C_VEL
LIN {X 0,Y 466.53,Z 521.145,A -85,B 0,C 180,E1 -7512.679,E2 -7512.679} C_VEL
LIN {X 0,Y 466.568,Z 521.031,A -85,B 0,C 180,E1 -7513.86,E2 -7513.86} C_VEL
LIN {X 0,Y 466.587,Z 520.143,A -85,B 0,C 180,E1 -7515.067,E2 -7515.067} C_VEL
LIN {X 0,Y 466.695,Z 517.411,A -85,B 0,C 180,E1 -7516.82,E2 -7516.82} C_VEL
LIN {X 0,Y 466.798,Z 514.521,A -85,B 0,C 180,E1 -7518.031,E2 -7518.031} C_VEL
LIN {X 0,Y 466.975,Z 509.136,A -85,B 0,C 180,E1 -7519.673,E2 -7519.673} C_VEL
LIN {X 0,Y 467.268,Z 502.567,A -85,B 0,C 180,E1 -7521.163,E2 -7521.163} C_VEL
LIN {X 0,Y 467.588,Z 495.681,A -85,B 0,C 180,E1 -7522.402,E2 -7522.402} C_VEL
LIN {X 0,Y 468.044,Z 486.347,A -85,B 0,C 180,E1 -7523.755,E2 -7523.755} C_VEL
LIN {X 0,Y 468.527,Z 476.815,A -85,B 0,C 180,E1 -7524.856,E2 -7524.856} C_VEL
LIN {X 0,Y 469.042,Z 466.591,A -85,B 0,C 180,E1 -7525.813,E2 -7525.813} C_VEL
LIN {X 0,Y 469.499,Z 454.982,A -85,B 0,C 180,E1 -7526.686,E2 -7526.686} C_VEL
LIN {X 0,Y 470.024,Z 442.798,A -85,B 0,C 180,E1 -7527.382,E2 -7527.382} C_VEL
LIN {X 0,Y 470.101,Z 433.033,A -85,B 0,C 180,E1 -7527.819,E2 -7527.819} C_VEL
LIN {X 0,Y 467.287,Z 420.148,A -85,B 0,C 180,E1 -7528.33,E2 -7528.33} C_VEL
LIN {X 0,Y 466.787,Z 417.849,A -85,B 0,C 180,E1 -7528.415,E2 -7528.415} C_VEL
LIN {X 0,Y 466.854,Z 414.05,A -85,B 0,C 180,E1 -7531.202,E2 -7531.202} C_VEL
LIN {X 0,Y 466.966,Z 410.111,A -85,B 0,C 180,E1 -7534.122,E2 -7534.122} C_VEL
LIN {X 0,Y 467.103,Z 406.349,A -85,B 0,C 180,E1 -7536.971,E2 -7536.971} C_VEL
LIN {X 0,Y 467.194,Z 402.702,A -85,B 0,C 180,E1 -7539.758,E2 -7539.758} C_VEL
LIN {X 0,Y 467.298,Z 399.199,A -85,B 0,C 180,E1 -7542.495,E2 -7542.495} C_VEL
LIN {X 0,Y 467.385,Z 395.811,A -85,B 0,C 180,E1 -7545.189,E2 -7545.189} C_VEL
LIN {X 0,Y 467.541,Z 392.524,A -85,B 0,C 180,E1 -7547.852,E2 -7547.852} C_VEL
LIN {X 0,Y 467.601,Z 392.244,A -85,B 0,C 180,E1 -7549.609,E2 -7549.609} C_VEL
LIN {X 0,Y 467.748,Z 392.224,A -85,B 0,C 180,E1 -7552.59,E2 -7552.59} C_VEL
LIN {X 0,Y 467.721,Z 392.226,A -85,B 0,C 180,E1 -7554.827,E2 -7554.827} C_VEL
LIN {X 0,Y 467.856,Z 392.21,A -85,B 0,C 180,E1 -7557.417,E2 -7557.417} C_VEL
LIN {X 0,Y 467.878,Z 392.206,A -85,B 0,C 180,E1 -7560,E2 -7560} C_VEL
LIN {X 0,Y 467.855,Z 392.208,A -85,B 0,C 180,E1 -7562.583,E2 -7562.583} C_VEL
LIN {X 0,Y 467.74,Z 392.225,A -85,B 0,C 180,E1 -7566.038,E2 -7566.038} C_VEL
LIN {X 0,Y 467.678,Z 392.231,A -85,B 0,C 180,E1 -7568.643,E2 -7568.643} C_VEL
LIN {X 0,Y 467.651,Z 392.235,A -85,B 0,C 180,E1 -7572.146,E2 -7572.146} C_VEL
LIN {X 0,Y 467.635,Z 392.236,A -85,B 0,C 180,E1 -7575.695,E2 -7575.695} C_VEL
LIN {X 0,Y 467.614,Z 392.239,A -85,B 0,C 180,E1 -7578.765,E2 -7578.765} C_VEL
LIN {X 0,Y 467.577,Z 392.243,A -85,B 0,C 180,E1 -7581.269,E2 -7581.269} C_VEL
LIN {X 0,Y 467.569,Z 392.242,A -85,B 0,C 180,E1 -7583.944,E2 -7583.944} C_VEL
LIN {X 0,Y 467.624,Z 392.239,A -85,B 0,C 180,E1 -7586.8,E2 -7586.8} C_VEL
LIN {X 0,Y 467.584,Z 392.244,A -85,B 0,C 180,E1 -7589.736,E2 -7589.736} C_VEL
LIN {X 0,Y 467.58,Z 392.244,A -85,B 0,C 180,E1 -7592.759,E2 -7592.759} C_VEL
LIN {X 0,Y 467.553,Z 392.248,A -85,B 0,C 180,E1 -7595.89,E2 -7595.89} C_VEL
LIN {X 0,Y 467.616,Z 392.241,A -85,B 0,C 180,E1 -7599.142,E2 -7599.142} C_VEL
LIN {X 0,Y 467.584,Z 392.244,A -85,B 0,C 180,E1 -7602.568,E2 -7602.568} C_VEL
LIN {X 0,Y 467.568,Z 392.245,A -85,B 0,C 180,E1 -7605.054,E2 -7605.054} C_VEL
LIN {X 0,Y 467.587,Z 392.244,A -85,B 0,C 180,E1 -7607.441,E2 -7607.441} C_VEL
LIN {X 0,Y 467.633,Z 392.333,A -85,B 0,C 180,E1 -7610.112,E2 -7610.112} C_VEL
LIN {X 0,Y 468.538,Z 398.019,A -85,B 0,C 180,E1 -7613.131,E2 -7613.131} C_VEL
LIN {X 0,Y 468.766,Z 402.393,A -85,B 0,C 180,E1 -7615.27,E2 -7615.27} C_VEL
LIN {X 0,Y 468.34,Z 409.07,A -85,B 0,C 180,E1 -7618.318,E2 -7618.318} C_VEL
LIN {X 0,Y 467.972,Z 415.901,A -85,B 0,C 180,E1 -7621.278,E2 -7621.278} C_VEL
LIN {X 0,Y 467.661,Z 423.327,A -85,B 0,C 180,E1 -7624.38,E2 -7624.38} C_VEL
LIN {X 0,Y 467.413,Z 430.961,A -85,B 0,C 180,E1 -7627.455,E2 -7627.455} C_VEL
LIN {X 0,Y 467.177,Z 438.002,A -85,B 0,C 180,E1 -7630.216,E2 -7630.216} C_VEL
LIN {X 0,Y 467.037,Z 446.279,A -85,B 0,C 180,E1 -7633.387,E2 -7633.387} C_VEL
LIN {X 0,Y 466.964,Z 449.485,A -85,B 0,C 180,E1 -7634.598,E2 -7634.598} C_VEL
LIN {X 0,Y 468.968,Z 462.85,A -85,B 0,C 180,E1 -7635.021,E2 -7635.021} C_VEL
LIN {X 0,Y 469.94,Z 471.389,A -85,B 0,C 180,E1 -7635.383,E2 -7635.383} C_VEL
LIN {X 0,Y 469.43,Z 484.41,A -85,B 0,C 180,E1 -7636.031,E2 -7636.031} C_VEL
LIN {X 0,Y 468.906,Z 495.836,A -85,B 0,C 180,E1 -7636.788,E2 -7636.788} C_VEL
LIN {X 0,Y 468.434,Z 506.774,A -85,B 0,C 180,E1 -7637.702,E2 -7637.702} C_VEL
LIN {X 0,Y 467.978,Z 516.849,A -85,B 0,C 180,E1 -7638.742,E2 -7638.742} C_VEL
LIN {X 0,Y 467.521,Z 525.415,A -85,B 0,C 180,E1 -7639.827,E2 -7639.827} C_VEL
LIN {X 0,Y 467.192,Z 533.769,A -85,B 0,C 180,E1 -7641.131,E2 -7641.131} C_VEL
LIN {X 0,Y 466.945,Z 540.509,A -85,B 0,C 180,E1 -7642.433,E2 -7642.433} C_VEL
LIN {X 0,Y 466.766,Z 546.687,A -85,B 0,C 180,E1 -7643.95,E2 -7643.95} C_VEL
LIN {X 0,Y 466.694,Z 550.701,A -85,B 0,C 180,E1 -7645.249,E2 -7645.249} C_VEL
LIN {X 0,Y 466.692,Z 553.671,A -85,B 0,C 180,E1 -7646.547,E2 -7646.547} C_VEL
LIN {X 0,Y 466.662,Z 555.085,A -85,B 0,C 180,E1 -7647.411,E2 -7647.411} C_VEL
LIN {X 0,Y 466.619,Z 556.717,A -85,B 0,C 180,E1 -7649.137,E2 -7649.137} C_VEL
LIN {X 0,Y 466.598,Z 556.941,A -85,B 0,C 180,E1 -7650,E2 -7650} C_VEL
LIN {X 0,Y 466.619,Z 556.73,A -85,B 0,C 180,E1 -7650.863,E2 -7650.863} C_VEL
LIN {X 0,Y 466.662,Z 555.131,A -85,B 0,C 180,E1 -7652.59,E2 -7652.59} C_VEL
LIN {X 0,Y 466.692,Z 553.729,A -85,B 0,C 180,E1 -7653.454,E2 -7653.454} C_VEL
LIN {X 0,Y 466.694,Z 550.78,A -85,B 0,C 180,E1 -7654.751,E2 -7654.751} C_VEL
LIN {X 0,Y 466.766,Z 546.784,A -85,B 0,C 180,E1 -7656.05,E2 -7656.05} C_VEL
LIN {X 0,Y 466.951,Z 540.632,A -85,B 0,C 180,E1 -7657.568,E2 -7657.568} C_VEL
